// POUs/Devices/CCU/FB_METIS_CCUS
FUNCTION_BLOCK FB_METIS_CCUS
VAR_INPUT
END_VAR
VAR_OUTPUT
END_VAR
VAR
    // Cabinet Control Units (note: CCU number is not linked to the cabinet number!!!)
    ccu_ns_1 : FB_MET_CCU;
    ccu_ns_2 : FB_MET_CCU;
    // ccu_ns_3 : FB_MET_CCU; // future
    // ccu_ns_4 : FB_MET_CCU; // future
    // ccu_ns_5 : FB_MET_CCU; // future
    // ccu_ns_6 : FB_MET_CCU; // future
    
    // simulators
    // ccu_ns_1_sim : FB_SIM_MET_CCU;
    // ccu_ns_2_sim : FB_SIM_MET_CCU;
    // ccu_ns_3_sim : FB_SIM_MET_CCU;
    // ccu_ns_4_sim : FB_SIM_MET_CCU; 
    // ccu_ns_5_sim : FB_SIM_MET_CCU;
    // ccu_ns_6_sim : FB_SIM_MET_CCU;
    
    // cooling config handlers
    {attribute 'OPC.UA.DA' := '0'}
    aCoolingConfig : ARRAY[1..2] OF FB_READ_WRITE_CAB_COOLING_CONFIG;
    
    // power config handlers
    {attribute 'OPC.UA.DA' := '0'}
    aPowerConfig : ARRAY[1..2] OF FB_READ_WRITE_CAB_POWER_CONFIG;
    
    // configure bool
    {attribute 'OPC.UA.DA' := '0'}
    bConfigured : BOOL;
END_VAR

// run the cooling config handlers (before configure!)
aCoolingConfig[1](in_sName := 'Cab_Cooling_1', stConfig := ccu_ns_1.cooling.cfg);
aCoolingConfig[2](in_sName := 'Cab_Cooling_2', stConfig := ccu_ns_2.cooling.cfg);
// aCoolingConfig[3](in_sName := 'Cab_Cooling_3', stConfig := ccu_ns_3.cooling.cfg); // future
// aCoolingConfig[4](in_sName := 'Cab_Cooling_4', stConfig := ccu_ns_4.cooling.cfg); // future
// aCoolingConfig[5](in_sName := 'Cab_Cooling_5', stConfig := ccu_ns_5.cooling.cfg); // future
// aCoolingConfig[6](in_sName := 'Cab_Cooling_6', stConfig := ccu_6.cooling.cfg); // future

// run the power config handlers (before configure!)
aPowerConfig[1](in_sName := 'Cab_Power_1', stConfig := ccu_ns_1.power.cfg);
aPowerConfig[2](in_sName := 'Cab_Power_2', stConfig := ccu_ns_2.power.cfg);
// aPowerConfig[3](in_sName := 'Cab_Power_3', stConfig := ccu_ns_3.power.cfg); // future
// aPowerConfig[4](in_sName := 'Cab_Power_4', stConfig := ccu_ns_4.power.cfg); // future
// aPowerConfig[5](in_sName := 'Cab_Power_5', stConfig := ccu_ns_5.power.cfg); // future
// aPowerConfig[6](in_sName := 'Cab_Power_6', stConfig := ccu_ns_6.power.cfg); // future

// run M_Configure *after* the config handlers above! 
IF NOT bConfigured THEN
    M_Configure();
    RETURN;
END_IF


// run the CCUs
ccu_ns_1(in_sCuName := 'CCU_NS_1', in_sCabinetName := 'Cabinet 6');
ccu_ns_2(in_sCuName := 'CCU_NS_2', in_sCabinetName := 'Cabinet 4');
// ccu_ns_3(in_sCuName := 'CCU_NS_3', in_sCabinetName := 'Cabinet TBD');
// ccu_ns_4(in_sCuName := 'CCU_NS_4', in_sCabinetName := 'Cabinet TBD');
// ccu_ns_5(in_sCuName := 'CCU_NS_5', in_sCabinetName := 'Cabinet TBD');
// ccu_ns_6(in_sCuName := 'CCU_NS_6', in_sCabinetName := 'Cabinet TBD');

// run the simulators for which no hardware is available yet
// ccu_ns_3_sim(ptrDev := ADR(ccu_ns_3));
// ccu_ns_4_sim(ptrDev := ADR(ccu_ns_4)); 
// ccu_ns_5_sim(ptrDev := ADR(ccu_ns_5));
// ccu_ns_6_sim(ptrDev := ADR(ccu_ns_6));

METHOD M_Configure : BOOL
VAR_INPUT
END_VAR
VAR_INST
	{attribute 'OPC.UA.DA' := '0'}
    nConfigureState : INT;
END_VAR
VAR_IN_OUT
	//{attribute 'OPC.UA.DA' := '0'}
END_VAR
VAR
    i : INT;
    bDone : BOOL;
    iMax : INT := 2;
END_VAR

CASE nConfigureState OF
    0:  ;
        
        // start reading the configs
        FOR i := 1 TO iMax DO
            aCoolingConfig[i].M_ReadConfiguration();
            aPowerConfig[i].M_ReadConfiguration();
        END_FOR
        nConfigureState := 1;
    1:
        bDone := TRUE;
        FOR i := 1 TO iMax DO
            IF NOT aCoolingConfig[i].bReadingDoneFlag THEN
                bDone := FALSE;
			END_IF
            IF NOT aPowerConfig[i].bReadingDoneFlag THEN
                bDone := FALSE;
			END_IF
        END_FOR
        IF bDone THEN
            nConfigureState := 2;
		END_IF
    2:
        FOR i := 1 TO iMax DO
            aCoolingConfig[i].M_ClearReadingDoneFlag();
            aPowerConfig[i].M_ClearReadingDoneFlag();
        END_FOR
        bConfigured := TRUE;
        
END_CASE
END_METHOD

END_FUNCTION_BLOCK

// POUs/XML_Cfg_Read_Write/FB_READ_WRITE_CAB_COOLING_CONFIG
FUNCTION_BLOCK FB_READ_WRITE_CAB_COOLING_CONFIG EXTENDS FB_READ_WRITE_CONFIG_BASE
VAR_INPUT
	in_sName:      T_MaxString;
END_VAR
VAR_IN_OUT
	stConfig:   T_CAB_COOLING_CFG;
END_VAR

SUPER^(
    in_sEntryName  := in_sName,
    in_sSubFolder  := 'Cab_Cooling\',
    in_sXPath      := '/Cab_Cooling_Configuration/',
    in_pSymAddr    := ADR(stConfig),
    in_cbSymSize   := SIZEOF(stConfig));

END_FUNCTION_BLOCK

// POUs/XML_Cfg_Read_Write/FB_READ_WRITE_CAB_POWER_CONFIG
FUNCTION_BLOCK FB_READ_WRITE_CAB_POWER_CONFIG EXTENDS FB_READ_WRITE_CONFIG_BASE
VAR_INPUT
	in_sName:      T_MaxString;
END_VAR
VAR_IN_OUT
	stConfig:   T_CAB_POWER_CFG;
END_VAR

SUPER^(
    in_sEntryName  := in_sName,
    in_sSubFolder  := 'Cab_Power\',
    in_sXPath      := '/Cab_Power_Configuration/',
    in_pSymAddr    := ADR(stConfig),
    in_cbSymSize   := SIZEOF(stConfig));

END_FUNCTION_BLOCK

// POUs/Routines/Evacuation/FB_METIS_CRYO_EVAC
FUNCTION_BLOCK FB_METIS_CRYO_EVAC
VAR_INPUT
	in_sName:							STRING := 'EVACUATION';
	in_Cryo_Stat:					T_METIS_CRYO_STAT;
END_VAR
VAR_IN_OUT
	{attribute 'OPC.UA.DA' := '0'}
	interlocks:						T_METIS_CRYO_INTERLOCKS;
END_VAR
VAR_OUTPUT
	out_bEvacuationActive:			BOOL;
END_VAR
VAR
	// Stat
	{attribute 'TcHmiSymbol.Show'}
	stat:							T_MET_CRYO_EVACUATION_STAT;
	// Ctrl
	{attribute 'TcHmiSymbol.Show'}
	ctrl:							T_MET_CRYO_EVACUATION_CTRL;
	// Evacuation-branch A
		{attribute 'TcHmiSymbol.Show'}
	evac_branch_a:		FB_CRYO_EVAC_BRANCH_A;
	// Evacuation-branch B
		{attribute 'TcHmiSymbol.Show'}
	evac_branch_b:		FB_CRYO_EVAC_BRANCH_B;

	
	bEnable_met_evac:	BOOL;
	
	bEnable_met_evac_a:	BOOL := FALSE;
	bEnable_met_evac_b:	BOOL := FALSE;
	
	// Pressure Sensors
	sensor_VAGF1:		FB_CRYO_SENSOR_PRESSURE;	// Cryo pressure gauge VAG F1
	VAGF1:				FB_CRYO_PRESSURE_VOTE;
	sensor_VAGF2:		FB_CRYO_SENSOR_PRESSURE;	// Cryo pressure gauge VAG F2
	VAGF2:				FB_CRYO_PRESSURE_VOTE;
	sensor_VAGG1:		FB_CRYO_SENSOR_PRESSURE;	// Cryo pressure gauge VAG G1
	VAGG1:				FB_CRYO_PRESSURE_VOTE;
	sensor_VAGG2:		FB_CRYO_SENSOR_PRESSURE;	// Cryo pressure gauge VAG G2
	VAGG2:				FB_CRYO_PRESSURE_VOTE;
	VAGF:				FB_CRYO_PRESSURE_VOTE;				// Cryo pressure F
	VAGG:				FB_CRYO_PRESSURE_VOTE;				// Cryo pressure G
	
	
	// Pressure sensors IDN resistors
	
	nIdnRes_VAG_F1		AT %I* :INT;
	nIdnRes_VAG_F2		AT %I* :INT;
	nIdnRes_VAG_G1		AT %I* :INT;
	nIdnRes_VAG_G2		AT %I* :INT;
	nIdnRes_VAG_A1		AT %I* :INT;
	nIdnRes_VAG_A2		AT %I* :INT;
	nIdnRes_VAG_A3		AT %I* :INT;
	nIdnRes_VAG_B1		AT %I* :INT;
	nIdnRes_VAG_B2		AT %I* :INT;
	nIdnRes_VAG_B3		AT %I* :INT;
	
	// Pressure sensor power 24V Dig Out
	
	bPwr_VAG_F1			AT %Q* :BOOL;
	bPwr_VAG_F2         AT %Q* :BOOL;
	bPwr_VAG_G1         AT %Q* :BOOL;
	bPwr_VAG_G2         AT %Q* :BOOL;
	bPwr_VAG_A1         AT %Q* :BOOL;
	bPwr_VAG_A2         AT %Q* :BOOL;
	bPwr_VAG_A3         AT %Q* :BOOL;
	bPwr_VAG_B1         AT %Q* :BOOL;
	bPwr_VAG_B2         AT %Q* :BOOL;
	bPwr_VAG_B3         AT %Q* :BOOL;
	
	// Valve Command handling
	cmdPVVA1:			FB_CRYO_ACTUATOR_CMD;
	bCmdPVVA1:			BOOL;	// Open/Close command for PVV1
	bIntlkPVVA1:		BOOL;	// Interlock for PVV1
	
	cmdPVVB1:			FB_CRYO_ACTUATOR_CMD;
	bCmdPVVB1:			BOOL;	// Open/Close command for PVV1
	bIntlkPVVB1:		BOOL;	// Interlock for PVV1
	
//	// Valve Power
//	bBrA_PVVs_Pwr					AT %Q* :BOOL;
//	bBrA_PVVs_FeedBack_Pwr			AT %Q* :BOOL;
//	bBrB_PVVs_Pwr					AT %Q* :BOOL;
//	bBrB_PVVs_FeedBack_Pwr			AT %Q* :BOOL;
//	bPVV_Ps_Pwr						AT %Q* :BOOL;
//	bPVV_Ps_FeedBack_Pwr			AT %Q* :BOOL;
//	bPCA_PCB_VV_Pwr					AT %Q* :BOOL;
//	bPCA_PCB_VV_FeedBack_Pwr		AT %Q* :BOOL;


	// Triggers.
	//
	// Capture Enable/Disable.
	trigAutoEnable:		R_TRIG;	// bEnable_met_evac
	trigAutoDisable:	F_TRIG;	// bEnable_met_evac
	
	trigManualEnable:		R_TRIG;	// ctrl.bEnable
	trigManualDisable:		F_TRIG;	// ctrl.bEnable

	

/////////////////////////////////////////////////////////////////////////////
////////////////// Simulation////////////////////////////////////////////////
/////////////////////////////////////////////////////////////////////////////
	
	met_valves_a:		FB_SIM_MICADO_VALVES;
	met_pumps_a:		FB_SIM_MICADO_PUMPS;
	
	met_valves_b:		FB_SIM_MICADO_VALVES;
	met_pumps_b:		FB_SIM_MICADO_PUMPS;
	
	// Pressure values
	q_nVAGA1			AT %Q*:	INT := 30000;
	q_nVAGA2			AT %Q*:	INT := 30000;
	q_nVAGA3			AT %Q*:	INT := 30000;
	
	q_nVAGB1			AT %Q*:	INT := 30000;
	q_nVAGB2			AT %Q*:	INT := 30000;
	q_nVAGB3			AT %Q*:	INT := 30000;
	
	q_nVAGF1			AT %Q*:	INT := 30000;
	q_nVAGF2			AT %Q*:	INT := 30000;
	q_nVAGG1			AT %Q*:	INT := 30000;
	q_nVAGG2			AT %Q*:	INT := 30000;
	
	// 230 VAC Power  for TMPs
	
	q_bTP_A_pwr			AT %Q*: BOOL;
	bTP_A_pwr: 					BOOL := TRUE;
	q_bTP_B_pwr			AT %Q*: BOOL;
	bTP_B_pwr: 					BOOL := TRUE;
	// Dig iuput 24V source
	q_bTP_A_Ready			AT %Q*: BOOL := FALSE;
	q_bTP_A_Speed100		AT %Q*: BOOL := FALSE;
	q_bTP_A_Warning			AT %Q*: BOOL := FALSE; 
	q_bTP_A_Error			AT %Q*: BOOL := FALSE;
	q_bTP_B_Ready			AT %Q*: BOOL := FALSE;
	q_bTP_B_Speed100		AT %Q*: BOOL := FALSE;
	q_bTP_B_Warning			AT %Q*: BOOL := FALSE; 
	q_bTP_B_Error			AT %Q*: BOOL := FALSE;
	
	// Used for simulated toggle signal
	pSim:				FB_CRYO_SIM_PRESSURE;
	
	q_nCouplerState		AT %Q*:	INT := 8;

	/////////////////////
	// Cryo System logs
	/////////////////////
		
	logs:	FB_CRYO_FUNCTION_LOG;

	
	// Configure
	bConfigured:			BOOL := FALSE;
END_VAR


IF stat.bManual THEN
	;
ELSE
	IF stat.bAuto THEN
		ctrl.bEnable := bEnable_met_evac;
		stat.bAuto := FALSE;
	ELSE
		;
	END_IF
END_IF

M_Configure();

M_HandleEvents();

M_ExecuteControllers();


M_HandleInterlocks();

M_UpdateStatus();

METHOD M_AreAnyPumpsRunning : BOOL
VAR_INPUT
END_VAR


//IF  evac_branch_a.tpRef.M_GetSpeed() = 0 AND   // speed of Turbo pump on branch A
//	evac_branch_a.rpRef.M_GetSpeed() = 0 AND  // speed of roughing on branch A
//	evac_branch_b.tpRef.M_GetSpeed() = 0 AND  // speed of Turbo pump on branch B
//	evac_branch_b.rpRef.M_GetSpeed() = 0 THEN  // speed of roughing on branch B
	
//	M_AreAnyPumpsRunning := FALSE;
	
//ELSE
//	M_AreAnyPumpsRunning := TRUE;
//END_IF


M_AreAnyPumpsRunning := evac_branch_a.tpRef.M_IsRunning() OR
						evac_branch_a.rpRef.M_IsRunning() OR
						evac_branch_b.tpRef.M_IsRunning() OR
						evac_branch_b.rpRef.M_IsRunning();
END_METHOD

METHOD M_AreRoughingPumpRunning : BOOL
VAR_INPUT
END_VAR


//IF 
//	evac_branch_a.rpRef.M_GetSpeed() = 0 AND  // speed of roughing on branch A	
//	evac_branch_b.rpRef.M_GetSpeed() = 0 THEN  // speed of roughing on branch B
	
//	M_AreRoughingPumpRunning := FALSE;
	
//ELSE
//	M_AreRoughingPumpRunning := TRUE;
//END_IF

M_AreRoughingPumpRunning := evac_branch_a.rpRef.M_IsRunning() AND evac_branch_b.rpRef.M_IsRunning();
END_METHOD

METHOD M_AreTurboPumpsRunning : BOOL
VAR_INPUT
END_VAR


//IF  evac_branch_a.tpRef.M_GetSpeed() = 0 AND   // speed of Turbo pump on branch A
//	evac_branch_b.tpRef.M_GetSpeed() = 0 THEN  // speed of Turbo pump on branch B

	
//	M_AreTurboPumpsRunning := FALSE;
	
//ELSE
//	M_AreTurboPumpsRunning := TRUE;
//END_IF


M_AreTurboPumpsRunning := evac_branch_a.tpRef.M_IsRunning() AND evac_branch_a.tpRef.M_IsRunning();
END_METHOD

METHOD M_CheckBranchError : BOOL
VAR_INPUT
END_VAR
//IF  evac_branch_a.tpRef.M_GetSpeed() = 0 AND   // speed of Turbo pump on branch A
//	evac_branch_a.rpRef.M_GetSpeed() = 0 AND  // speed of roughing on branch A
//	evac_branch_b.tpRef.M_GetSpeed() = 0 AND  // speed of Turbo pump on branch B
//	evac_branch_b.rpRef.M_GetSpeed() = 0 THEN  // speed of roughing on branch B


// evac_branch_a.stat.bError
END_METHOD

METHOD M_Configure
VAR_INPUT
END_VAR
IF NOT bConfigured THEN
	

	// Enable Pressure sensor power
	bPwr_VAG_F1		 :=	TRUE;																				
	bPwr_VAG_F2      :=	TRUE;
	bPwr_VAG_G1      :=	TRUE;
	bPwr_VAG_G2      :=	TRUE;
	bPwr_VAG_A1      :=	TRUE;
	bPwr_VAG_A2      :=	TRUE;
	bPwr_VAG_A3      :=	TRUE;
	bPwr_VAG_B1      :=	TRUE;
	bPwr_VAG_B2      :=	TRUE;
	bPwr_VAG_B3      :=	TRUE;


//Enable power for valves, feedback of the valves
//	bBrA_PVVs_Pwr						:=	TRUE;	
//    bBrA_PVVs_FeedBack_Pwr	            :=	TRUE;
//    bBrB_PVVs_Pwr			            :=	TRUE;
//    bBrB_PVVs_FeedBack_Pwr	            :=	TRUE;
//    bPVV_Ps_Pwr				            :=	TRUE;
//    bPVV_Ps_FeedBack_Pwr	            :=	TRUE;
//    bPCA_PCB_VV_Pwr			            :=	TRUE;
//    bPCA_PCB_VV_FeedBack_Pwr            :=	TRUE;


	
	
	q_bTP_A_Ready	 := TRUE;
	q_bTP_A_Speed100 := TRUE;
	q_bTP_A_Warning	 := TRUE;
	q_bTP_A_Error	 := TRUE;
	q_bTP_B_Ready	 := TRUE;
	q_bTP_B_Speed100 := TRUE;
	q_bTP_B_Warning	 := TRUE;
	q_bTP_B_Error	 := TRUE;
	
// This call just configures logs at the very start.
// Logging is done by explicit calls to M_LogInfo().
logs(in_sName := in_sName);	

                                   
	bConfigured := TRUE;
END_IF
END_METHOD

METHOD M_ExecuteControllers
VAR_INPUT
END_VAR

// 230 VAC Power  for TMPs

	q_bTP_A_pwr := bTP_A_pwr;
    q_bTP_B_pwr := bTP_B_pwr;

// METIS Cryostat pressures
sensor_VAGF1(in_sName := 'VAGF1' ,in_nType := E_CRYO_SENSOR_TYPE_PRESS.PKR_360,	in_nSampleTime := 100);
sensor_VAGF2(in_sName := 'VAGF2' ,in_nType := E_CRYO_SENSOR_TYPE_PRESS.PKR_360,	in_nSampleTime := 100);
sensor_VAGG1(in_sName := 'VAGG1' ,in_nType := E_CRYO_SENSOR_TYPE_PRESS.PKR_360,	in_nSampleTime := 100);
sensor_VAGG2(in_sName := 'VAGG2' ,in_nType := E_CRYO_SENSOR_TYPE_PRESS.PKR_360,	in_nSampleTime := 100);


ctrl.por_VAGF1(in_bEnable := ctrl.bSim_Press_VAGF1);	// Simulation flag override
VAGF1(
	in_sName		:= 'VAGF1',
	in_bSimulation	:= ctrl.por_VAGF1.out_bEnable,
	in_nNumSensor	:= 1,
	in_nVoteMethod	:= E_CRYO_VOTE.V_AVE,
	in_pSensor1		:= ADR(sensor_VAGF1));

ctrl.por_VAGF2(in_bEnable := ctrl.bSim_Press_VAGF2);	// Simulation flag override
VAGF2(
	in_sName		:= 'VAGF2',
	in_bSimulation	:= ctrl.por_VAGF2.out_bEnable,
	in_nNumSensor	:= 1,
	in_nVoteMethod	:= E_CRYO_VOTE.V_AVE,
	in_pSensor1		:= ADR(sensor_VAGF2));

ctrl.por_VAGG1(in_bEnable := ctrl.bSim_Press_VAGG1);	// Simulation flag override
VAGG1(
	in_sName		:= 'VAGG1',
	in_bSimulation	:= ctrl.por_VAGG1.out_bEnable,
	in_nNumSensor	:= 1,
	in_nVoteMethod	:= E_CRYO_VOTE.V_AVE,
	in_pSensor1		:= ADR(sensor_VAGG1));

ctrl.por_VAGG2(in_bEnable := ctrl.bSim_Press_VAGG2);	// Simulation flag override
VAGG2(
	in_sName		:= 'VAGG2',
	in_bSimulation	:= ctrl.por_VAGG2.out_bEnable,
	in_nNumSensor	:= 1,
	in_nVoteMethod	:= E_CRYO_VOTE.V_AVE,
	in_pSensor1		:= ADR(sensor_VAGG2));

ctrl.por_VAGF(in_bEnable := ctrl.bSim_Press_VAGF);	// Simulation flag override
VAGF(
	in_sName		:= 'VAGF',
	in_bSimulation	:= ctrl.por_VAGF.out_bEnable,
	in_nNumSensor	:= 2,
	in_nVoteMethod	:= E_CRYO_VOTE.V_1oo2,
	in_pSensor1		:= ADR(sensor_VAGF1),
	in_pSensor2		:= ADR(sensor_VAGF2));
	
ctrl.por_VAGG(in_bEnable := ctrl.bSim_Press_VAGG);	// Simulation flag override
VAGG(
	in_sName		:= 'VAGG',
	in_bSimulation	:= ctrl.por_VAGG.out_bEnable,
	in_nNumSensor	:= 2,
	in_nVoteMethod	:= E_CRYO_VOTE.V_1oo2,
	in_pSensor1		:= ADR(sensor_VAGG1),
	in_pSensor2		:= ADR(sensor_VAGG2));
	
	
	
	
	
	
	
	
	

	
// METIS evacuation system
cmdPVVA1(in_bEnable:=bCmdPVVA1,in_bInterlock:=bIntlkPVVA1);	// Handling of PVV1 commands
cmdPVVB1(in_bEnable:=bCmdPVVB1,in_bInterlock:=bIntlkPVVB1);	// Handling of PVV1 commands


IF ctrl.bEnable THEN
	bEnable_met_evac_a := TRUE;
	bEnable_met_evac_b := TRUE;
ELSE
	bEnable_met_evac_a := FALSE;
	bEnable_met_evac_b := FALSE;
END_IF

evac_branch_a(
	in_bEnable		:= bEnable_met_evac_a,
	in_RefVAGF		:= VAGF, 
	in_RefVAGG		:= VAGG);

evac_branch_b(
	in_bEnable		:= bEnable_met_evac_a,
	in_RefVAGF		:= VAGF, 
	in_RefVAGG		:= VAGG);
	
	
	
{IF defined (V2_SIM)}
	{info 'Simulated valves'}	

pSim();	// Just to have a simulated Toggle signal.

// Simulation of METIS valves
met_valves_a();
met_valves_b();	

// Simulation of METIS pumps
met_pumps_a(in_RefPVP:=evac_branch_a.rp, in_RefTMP:=evac_branch_a.tp);	
met_pumps_b(in_RefPVP:=evac_branch_b.rp, in_RefTMP:=evac_branch_b.tp);	

{END_IF}
END_METHOD

METHOD M_HandleEvents
VAR_INPUT
END_VAR
VAR_INST
    nEvacOnOffState : UINT := 0; // 0=Idle, 10=AutoOn, 20=AutoOff, 30=ManualOn, 40=ManualOff
END_VAR

trigAutoEnable    (CLK := bEnable_met_evac);
trigAutoDisable   (CLK := bEnable_met_evac); 

trigManualEnable  (CLK := ctrl.bEnable);
trigManualDisable (CLK := ctrl.bEnable);


CASE nEvacOnOffState OF

    0: // Idle / waiting for an event
        IF trigAutoEnable.Q THEN
            nEvacOnOffState := 10;
        ELSIF trigAutoDisable.Q THEN
            nEvacOnOffState := 20;
        ELSIF trigManualEnable.Q THEN
            nEvacOnOffState := 30;
        ELSIF trigManualDisable.Q THEN
            nEvacOnOffState := 40;
        END_IF

    10: // Auto Enable event
        stat.sState := 'EVACUATION started automatically';
        logs.M_LogInfo('EVACUATION started automatically');
		M_ResetValves();
        nEvacOnOffState := 0; // back to idle

    20: // Auto Disable event
        stat.sState := 'EVACUATION stopped automatically';
        logs.M_LogInfo('EVACUATION stopped automatically');
		M_ResetValves();
        nEvacOnOffState := 0;

    30: // Manual Enable event
        stat.sState := 'EVACUATION started by operator';
        logs.M_LogInfo('EVACUATION started by operator');
		M_ResetValves();
        nEvacOnOffState := 0;

    40: // Manual Disable event
        stat.sState := 'EVACUATION interrupted by operator';
        logs.M_LogInfo('EVACUATION interrupted by operator');
		M_ResetValves();
        nEvacOnOffState := 0;

END_CASE
END_METHOD

METHOD M_HandleInterlocks
VAR_INPUT
END_VAR
END_METHOD

METHOD M_ResetValves : BOOL
VAR_INPUT
END_VAR
evac_branch_a.M_ResetValves();
evac_branch_b.M_ResetValves();
END_METHOD

METHOD M_SetAuto : BOOL
VAR_INPUT
END_VAR
stat.bAuto := TRUE;
END_METHOD

METHOD PRIVATE M_SetError
VAR_INPUT
    nCode     : UDINT;
    sMessage  : STRING;
END_VAR


stat.Error.nCode := nCode;
stat.Error.sMessage := sMessage;
stat.bError := TRUE;
//stat.nState := E_MET_CRYO_EVA.ERROR;
END_METHOD

METHOD M_Start_Evacuation : BOOL
VAR_INPUT
END_VAR
stat.bAuto := TRUE;
bEnable_met_evac := TRUE;
END_METHOD

METHOD M_Stop_Evacuation : BOOL
VAR_INPUT
END_VAR

stat.bAuto := TRUE;
bEnable_met_evac := FALSE;
END_METHOD

METHOD M_UpdateStatus
VAR_INPUT
END_VAR


// Check Pre-Conditions for HMI Enable 

stat.bPreConditionsMet :=  in_Cryo_Stat.bVentingValvesAreClosed;


stat.bActive := ctrl.bEnable;
out_bEvacuationActive := stat.bActive;

stat.bBusy := stat.bActive;
stat.bDone := NOT stat.bActive;
END_METHOD

END_FUNCTION_BLOCK

// POUs/Routines/Evacuation/FB_CRYO_EVAC_BRANCH_A
FUNCTION_BLOCK FB_CRYO_EVAC_BRANCH_A EXTENDS FB_CRYO_EVAC_BASE_50000
VAR_INPUT
END_VAR
VAR_OUTPUT
END_VAR
VAR
	// Specify pumps
	{attribute 'TcHmiSymbol.Show'}
	rp:				FB_CRYO_PUMP_ECODRY;	// Roughing Pump
	{attribute 'TcHmiSymbol.Show'}
	tp:				FB_CRYO_PUMP_ATH2303M;	// Turbomolecular Pump
	
	// Pumps command handeling
	cor_rp:			FB_CRYO_CMD_OVERRIDE;
	cor_tp:			FB_CRYO_CMD_OVERRIDE;
	
	
	
	bReset_Valves:		BOOL:= FALSE;
	
	
END_VAR






SUPER^();	// Execute base FB code.

IF bReset_Valves THEN
	M_ResetValves();
	bReset_Valves := FALSE;
END_IF

METHOD M_Configure
VAR_INPUT
END_VAR
//
// Specific METIS configuration.
//
IF NOT stat.bConfigured	THEN
	//
	// MANDATORY !!!
	// Call base FB::M_Configure() to set the pointers.
	//
	SUPER^.M_Configure();
	

	// MANDATORY: Set References for pumps!!!
	// If not done, system will crash !!!
	rpRef	REF=rp;
	tpRef	REF=tp;
	

	// Specific instance configuration, e.g. anything different
	// from the default values given in the cfg structure of type T_CRYO_EVAC_CFG_50000.
	cfg.nType_VAG1	:= E_CRYO_SENSOR_TYPE_PRESS.PKR_360;
	cfg.nType_VAG2	:= E_CRYO_SENSOR_TYPE_PRESS.PKR_360;
	cfg.nType_VAG3	:= E_CRYO_SENSOR_TYPE_PRESS.PKR_360;
	
	cfg.nType_VAGF1	:= E_CRYO_SENSOR_TYPE_PRESS.PKR_360;
	cfg.nType_VAGF2	:= E_CRYO_SENSOR_TYPE_PRESS.PKR_360;
	cfg.nType_VAGG1	:= E_CRYO_SENSOR_TYPE_PRESS.PKR_360;
	cfg.nType_VAGG2	:= E_CRYO_SENSOR_TYPE_PRESS.PKR_360;
	
	// Prevacuum pressure threshold [mbar]: TMP start below this 
	
	cfg.lrThld_Prevac:= 0.5;	 	

// Reseting all valves. Without this, the valves were not initializing in error and were unable to recover
	PVV1.M_Reset();
	PVV2.M_Reset();
	PVV3.M_Reset();
	PVV4.M_Reset();
	GBV.M_Reset();
	
	
	stat.bConfigured	:= TRUE;
ELSE
	RETURN;	// Nothing to do any more
END_IF
END_METHOD

METHOD M_ExecuteControllers
VAR_INPUT
END_VAR
// Pumps command overide 

cor_rp(in_bEnable:= ctrl.bEnable_PVP);
cor_tp(in_bEnable:= ctrl.bEnable_TMP);


{IF defined (V2_SIM)}
	{info 'Simulated Pumps'}
	
		// Roughing Pump	
	rp(	
		in_bSimulation	:= TRUE,
		in_sName		:= 'ECODRY A',
		in_bEnable		:= cor_rp.out_bEnable,
		in_nSlaveID		:= 1,
		in_sVersion		:= 'V22',
		in_nPeriod		:= 2000,
		in_bFeedbackActiveLow := TRUE			// TRUE for simulation and FALSE for real hardware		
	);
	
	// Turbo Molecular Pump
	tp(	
		in_bSimulation	:= TRUE,
		in_sName		:= 'ATH2303M A',
		in_bEnable		:= cor_tp.out_bEnable,
		in_nModel		:= 2303,
		in_bAutoMonitor	:= TRUE,
		in_nPeriod		:= 2000);
{END_IF}



{IF defined (V1_HW)}
	{info 'Actual Pumps are Active'}
	
		// Roughing Pump	
	rp(	
		in_bSimulation	:= FALSE,
		in_sName		:= 'ECODRY A',
		in_bEnable		:= cor_rp.out_bEnable,
		in_nSlaveID		:= 1,
		in_sVersion		:= 'V22',
		in_nPeriod		:= 2000,
		in_bFeedbackActiveLow := FALSE			// TRUE for simulation and FALSE for real hardware		
	);
	
	// Turbo Molecular Pump
	tp(	
		in_bSimulation	:= FALSE,
		in_sName		:= 'ATH2303M A',
		in_bEnable		:= cor_tp.out_bEnable,
		in_nModel		:= 2303,
		in_bAutoMonitor	:= TRUE,
		in_nPeriod		:= 2000);

{END_IF}





SUPER^.M_ExecuteControllers();
END_METHOD

METHOD M_HandleInterlocks
VAR_INPUT
END_VAR
////////////////////////////////////////////////////////////////////
// IMPORTANT NOTE !!!
//
// The naming of valves and pumps is in accordance with
// the official ESO document 
// Sequences for vacuum vessel 2500 - 50000L by Marcus v5.pdf.
//
// MICADO names are different/swapped.
//
/////////////////////////////////////////////////////////////////////


///////////////////////////////////////////
// Translation Table MICADO --> ESO Naming
///////////////////////////////////////////
(*
MPA-A-PVP	PVP
MPA-A-TMP	TMP

MPA-A-GBV	GBV
MPA-A-PVV1	PVV3
MPA-A-PVV2	PVV4
MPA-A-PVV3	PVV1
MPA-A-PVV4	PVV2

TMPA-A-VAG1	VAG3
TMPA-A-VAG2	VAG2
TMPA-A-VAG3	VAG1

WRGA-A-VAG	VAGF
WRGA-B-VAG	VAGG
*)


//////////////////////////////////////////
////////////     VALVES       ////////////
//////////////////////////////////////////


//				
// TMPA-A-GBV: Can only be opened IF TMPA-A-PVP is ON.
//----------------------------------------
// GBV: Can only be opened IF PVP is ON.
//
IF rp.stat.bMoving	THEN
	ctrl.cor_GBV.M_SetAllPermitted();			// OPEN/CLOSE allowed.
ELSE
	ctrl.cor_GBV.M_SetPermissions(FALSE,TRUE);	// Only CLOSE allowed.
END_IF


//
// TMPA-A-PVV3: Can only be opened if:
// 	i. TMPA-A-VAG1 is less than 10-1 mbar
// 	ii. TMPA-A-TMP is OFF
// 	iii. WRGA-A-VAG and WRGA-B-VAG show pressure readings greater than 10-1 mbar.
//----------------------------------------
// PVV1: Can only be opened if:
// 	i. VAG3 is less than 10-1 mbar
// 	ii. TMP is OFF
// 	iii. VAGF and VAGG show pressure readings greater than 10-1 mbar.
//
IF	VAG3.stat.lrPressure < 0.1  AND  
	NOT tp.stat.bSpeed100  		AND 
	VAGF.stat.lrPressure > 0.1  AND 
	VAGG.stat.lrPressure > 0.1		THEN
	ctrl.cor_PVV1.M_SetAllPermitted();			// OPEN/CLOSE allowed.
ELSE
	ctrl.cor_PVV1.M_SetPermissions(FALSE,TRUE);	// Only CLOSE allowed.
END_IF


//
//	TMPA-A-PVV4: Can only be opened if:
// 	i. TMPA-A-VAG1 and TMPA-A-VAG3 show pressure readings of less than 10-1mbar
// 	ii. TMPA-A-TMP is OFF
// 	iii. WRGA-A-VAG and WRGA-B-VAG show pressure readings greater than 10-1mbar.
//----------------------------------------
//	PVV2: Can only be opened if:
// 	i. TMPA-A-VAG3 and TMPA-A-VAG1 show pressure readings of less than 10-1 mbar
// 	ii. TMP is OFF
// 	iii. VAGF and VAGG show pressure readings greater than 10-1 mbar.
//
IF	VAG3.stat.lrPressure < 0.1  AND  
	VAG1.stat.lrPressure < 0.1  AND  
	NOT tp.stat.bSpeed100  		AND 
	VAGF.stat.lrPressure > 0.1  AND 
	VAGG.stat.lrPressure > 0.1		THEN
	ctrl.cor_PVV2.M_SetAllPermitted();			// OPEN/CLOSE allowed.
ELSE
	ctrl.cor_PVV2.M_SetPermissions(FALSE,TRUE);	// Only CLOSE allowed.
END_IF


//
// TMPA-A-PVV1: Can only be opened if TMPA-A-TMP is ON or TMPA-A-PVV2 is closed.
//----------------------------------------
// PVV3: Can only be opened if TMP is ON or PVV4 is closed.
//
IF tp.stat.bSpeed100  OR  PVV4.stat.bActOFF	THEN
	ctrl.cor_PVV3.M_SetAllPermitted();			// OPEN/CLOSE allowed.
ELSE
	ctrl.cor_PVV3.M_SetPermissions(FALSE,TRUE);	// Only CLOSE allowed.
END_IF


//
// TMPA-A-PVV2: Can only be opened if TMPA-A-VAG1 and TMPA-A-VAG2 show pressure readings below 10-1 mbar
//----------------------------------------
// PVV4: Can only be opened if VAG3 and VAG2 show pressure readings below 10-1 mbar
//
IF VAG3.stat.lrPressure < 0.1  AND  VAG2.stat.lrPressure < 0.1	THEN
	ctrl.cor_PVV4.M_SetAllPermitted();			// OPEN/CLOSE allowed.
ELSE
	ctrl.cor_PVV4.M_SetPermissions(FALSE,TRUE);	// Only CLOSE allowed.
END_IF



//////////////////////////////////////////
////////////     PUMPS        ////////////
//////////////////////////////////////////


//
// TMPA-A-PVP: No interlock.
//----------------------------------------
// PVP: No interlock.
//
ctrl.cor_PVP.M_SetAllPermitted();	// ON/OFF allowed.


//
// TMPA-A-TMP: Can only be switched ON if WRGA-A-VAG and WRGA-B-VAG show pressure readings below 10-1 mbar
//----------------------------------------
// TMP: Can only be switched ON if VAGF and VAGG show pressure readings below 10-1 mbar
//
IF	VAGF.stat.lrPressure < (0.1 + cfg.lrThld_PrevacTol) AND 
	VAGG.stat.lrPressure < (0.1 + cfg.lrThld_PrevacTol)		THEN
	ctrl.cor_TMP.M_SetAllPermitted();			// ON/OFF allowed.
ELSE
	ctrl.cor_TMP.M_SetPermissions(FALSE,TRUE);	// Only OFF allowed.
END_IF
END_METHOD

METHOD M_ResetValves
VAR_INPUT
END_VAR
PVV1.M_Reset();
PVV2.M_Reset();
PVV3.M_Reset();
PVV4.M_Reset();
GBV.M_Reset();
END_METHOD

END_FUNCTION_BLOCK

// POUs/Routines/Evacuation/FB_CRYO_EVAC_BRANCH_B
FUNCTION_BLOCK FB_CRYO_EVAC_BRANCH_B EXTENDS FB_CRYO_EVAC_BASE_50000
VAR_INPUT
END_VAR
VAR_OUTPUT
END_VAR
VAR
	// Specify pumps
	{attribute 'TcHmiSymbol.Show'}
	rp:				FB_CRYO_PUMP_ECODRY;	// Roughing Pump
	{attribute 'TcHmiSymbol.Show'}
	tp:				FB_CRYO_PUMP_ATH2303M;	// Turbomolecular Pump
	
	// Pumps command handeling
	cor_rp:			FB_CRYO_CMD_OVERRIDE;
	cor_tp:			FB_CRYO_CMD_OVERRIDE;
	
	
		bReset_Valves:		BOOL:= FALSE;
		
END_VAR

SUPER^();	// Execute base FB code.

IF bReset_Valves THEN
	M_ResetValves();
	bReset_Valves := FALSE;
END_IF

METHOD M_Configure
VAR_INPUT
END_VAR
//
// Specific MICADO configuration.
//
IF NOT stat.bConfigured	THEN
	//
	// MANDATORY !!!
	// Call base FB::M_Configure() to set the pointers.
	//
	SUPER^.M_Configure();
	

	// MANDATORY: Set References for pumps!!!
	// If not done, system will crash !!!
	rpRef	REF=rp;
	tpRef	REF=tp;
	

	// Specific instance configuration, e.g. anything different
	// from the default values given in the cfg structure of type T_CRYO_EVAC_CFG_50000.
	cfg.nType_VAG1	:= E_CRYO_SENSOR_TYPE_PRESS.PKR_360;
	cfg.nType_VAG2	:= E_CRYO_SENSOR_TYPE_PRESS.PKR_360;
	cfg.nType_VAG3	:= E_CRYO_SENSOR_TYPE_PRESS.PKR_360;
	cfg.nType_VAGF1	:= E_CRYO_SENSOR_TYPE_PRESS.PKR_360;
	cfg.nType_VAGF2	:= E_CRYO_SENSOR_TYPE_PRESS.PKR_360;
	cfg.nType_VAGG1	:= E_CRYO_SENSOR_TYPE_PRESS.PKR_360;
	cfg.nType_VAGG2	:= E_CRYO_SENSOR_TYPE_PRESS.PKR_360;
	
	// Prevacuum pressure threshold [mbar]: TMP start below this 
	
	cfg.lrThld_Prevac:= 0.5;	 

// Reseting all valves. Without this, the valves were not initializing in error and were unable to recover
	PVV1.M_Reset();
	PVV2.M_Reset();
	PVV3.M_Reset();
	PVV4.M_Reset();
	GBV.M_Reset();
	
	stat.bConfigured	:= TRUE;
ELSE
	RETURN;	// Nothing to do any more
END_IF
END_METHOD

METHOD M_ExecuteControllers
VAR_INPUT
END_VAR
// Pumps command overide 

cor_rp(in_bEnable:= ctrl.bEnable_PVP);
cor_tp(in_bEnable:= ctrl.bEnable_TMP);


{IF defined (V2_SIM)}
	{info 'Simulated Pumps'}
	
		// Roughing Pump	
	rp(	
		in_bSimulation	:= TRUE,
		in_sName		:= 'ECODRY B',
		in_bEnable		:= cor_rp.out_bEnable,
		in_nSlaveID		:= 1,
		in_sVersion		:= 'V22',
		in_nPeriod		:= 2000,
		in_bFeedbackActiveLow := TRUE			// TRUE for simulation and FALSE for real hardware		
	);
	
	// Turbo Molecular Pump
	tp(	
		in_bSimulation	:= TRUE,
		in_sName		:= 'ATH2303M B',
		in_bEnable		:= cor_tp.out_bEnable,
		in_nModel		:= 2303,
		in_bAutoMonitor	:= TRUE,
		in_nPeriod		:= 2000);
{END_IF}



{IF defined (V1_HW)}
	{info 'Actual Pumps are Active'}
	
		// Roughing Pump	
	rp(	
		in_bSimulation	:= FALSE,
		in_sName		:= 'ECODRY B',
		in_bEnable		:= cor_rp.out_bEnable,
		in_nSlaveID		:= 1,
		in_sVersion		:= 'V22',
		in_nPeriod		:= 2000,
		in_bFeedbackActiveLow := FALSE			// TRUE for simulation and FALSE for real hardware		
	);
	
	// Turbo Molecular Pump
	tp(	
		in_bSimulation	:= FALSE,
		in_sName		:= 'ATH2303M B',
		in_bEnable		:= cor_tp.out_bEnable,
		in_nModel		:= 2303,
		in_bAutoMonitor	:= TRUE,
		in_nPeriod		:= 2000);

{END_IF}





SUPER^.M_ExecuteControllers();
END_METHOD

METHOD M_HandleInterlocks
VAR_INPUT
END_VAR
////////////////////////////////////////////////////////////////////
// IMPORTANT NOTE !!!
//
// The naming of valves and pumps is in accordance with
// the official ESO document 
// Sequences for vacuum vessel 2500 - 50000L by Marcus v5.pdf.
//
// MICADO names are different/swapped.
//
/////////////////////////////////////////////////////////////////////


///////////////////////////////////////////
// Translation Table MICADO --> ESO Naming
///////////////////////////////////////////
(*
MPA-A-PVP	PVP
MPA-A-TMP	TMP

MPA-A-GBV	GBV
MPA-A-PVV1	PVV3
MPA-A-PVV2	PVV4
MPA-A-PVV3	PVV1
MPA-A-PVV4	PVV2

TMPA-A-VAG1	VAG3
TMPA-A-VAG2	VAG2
TMPA-A-VAG3	VAG1

WRGA-A-VAG	VAGF
WRGA-B-VAG	VAGG
*)


//////////////////////////////////////////
////////////     VALVES       ////////////
//////////////////////////////////////////


//				
// TMPA-A-GBV: Can only be opened IF TMPA-A-PVP is ON.
//----------------------------------------
// GBV: Can only be opened IF PVP is ON.
//
IF rp.stat.bMoving	THEN
	ctrl.cor_GBV.M_SetAllPermitted();			// OPEN/CLOSE allowed.
ELSE
	ctrl.cor_GBV.M_SetPermissions(FALSE,TRUE);	// Only CLOSE allowed.
END_IF


//
// TMPA-A-PVV3: Can only be opened if:
// 	i. TMPA-A-VAG1 is less than 10-1 mbar
// 	ii. TMPA-A-TMP is OFF
// 	iii. WRGA-A-VAG and WRGA-B-VAG show pressure readings greater than 10-1 mbar.
//----------------------------------------
// PVV1: Can only be opened if:
// 	i. VAG3 is less than 10-1 mbar
// 	ii. TMP is OFF
// 	iii. VAGF and VAGG show pressure readings greater than 10-1 mbar.
//
IF	VAG3.stat.lrPressure < 0.1  AND  
	NOT tp.stat.bSpeed100  		AND 
	VAGF.stat.lrPressure > 0.1  AND 
	VAGG.stat.lrPressure > 0.1		THEN
	ctrl.cor_PVV1.M_SetAllPermitted();			// OPEN/CLOSE allowed.
ELSE
	ctrl.cor_PVV1.M_SetPermissions(FALSE,TRUE);	// Only CLOSE allowed.
END_IF


//
//	TMPA-A-PVV4: Can only be opened if:
// 	i. TMPA-A-VAG1 and TMPA-A-VAG3 show pressure readings of less than 10-1mbar
// 	ii. TMPA-A-TMP is OFF
// 	iii. WRGA-A-VAG and WRGA-B-VAG show pressure readings greater than 10-1mbar.
//----------------------------------------
//	PVV2: Can only be opened if:
// 	i. TMPA-A-VAG3 and TMPA-A-VAG1 show pressure readings of less than 10-1 mbar
// 	ii. TMP is OFF
// 	iii. VAGF and VAGG show pressure readings greater than 10-1 mbar.
//
IF	VAG3.stat.lrPressure < 0.1  AND  
	VAG1.stat.lrPressure < 0.1  AND  
	NOT tp.stat.bSpeed100  		AND 
	VAGF.stat.lrPressure > 0.1  AND 
	VAGG.stat.lrPressure > 0.1		THEN
	ctrl.cor_PVV2.M_SetAllPermitted();			// OPEN/CLOSE allowed.
ELSE
	ctrl.cor_PVV2.M_SetPermissions(FALSE,TRUE);	// Only CLOSE allowed.
END_IF


//
// TMPA-A-PVV1: Can only be opened if TMPA-A-TMP is ON or TMPA-A-PVV2 is closed.
//----------------------------------------
// PVV3: Can only be opened if TMP is ON or PVV4 is closed.
//
IF tp.stat.bSpeed100  OR  PVV4.stat.bActOFF	THEN
	ctrl.cor_PVV3.M_SetAllPermitted();			// OPEN/CLOSE allowed.
ELSE
	ctrl.cor_PVV3.M_SetPermissions(FALSE,TRUE);	// Only CLOSE allowed.
END_IF


//
// TMPA-A-PVV2: Can only be opened if TMPA-A-VAG1 and TMPA-A-VAG2 show pressure readings below 10-1 mbar
//----------------------------------------
// PVV4: Can only be opened if VAG3 and VAG2 show pressure readings below 10-1 mbar
//
IF VAG3.stat.lrPressure < 0.1  AND  VAG2.stat.lrPressure < 0.1	THEN
	ctrl.cor_PVV4.M_SetAllPermitted();			// OPEN/CLOSE allowed.
ELSE
	ctrl.cor_PVV4.M_SetPermissions(FALSE,TRUE);	// Only CLOSE allowed.
END_IF



//////////////////////////////////////////
////////////     PUMPS        ////////////
//////////////////////////////////////////


//
// TMPA-A-PVP: No interlock.
//----------------------------------------
// PVP: No interlock.
//
ctrl.cor_PVP.M_SetAllPermitted();	// ON/OFF allowed.


//
// TMPA-A-TMP: Can only be switched ON if WRGA-A-VAG and WRGA-B-VAG show pressure readings below 10-1 mbar
//----------------------------------------
// TMP: Can only be switched ON if VAGF and VAGG show pressure readings below 10-1 mbar
//
IF	VAGF.stat.lrPressure < (0.1 + cfg.lrThld_PrevacTol) AND 
	VAGG.stat.lrPressure < (0.1 + cfg.lrThld_PrevacTol)		THEN
	ctrl.cor_TMP.M_SetAllPermitted();			// ON/OFF allowed.
ELSE
	ctrl.cor_TMP.M_SetPermissions(FALSE,TRUE);	// Only OFF allowed.
END_IF
END_METHOD

METHOD M_ResetValves
VAR_INPUT
END_VAR
PVV1.M_Reset();
PVV2.M_Reset();
PVV3.M_Reset();
PVV4.M_Reset();
GBV.M_Reset();
END_METHOD

END_FUNCTION_BLOCK

// POUs/Routines/Venting/FB_METIS_CRYO_VENTING
FUNCTION_BLOCK FB_METIS_CRYO_VENTING
VAR_INPUT
	in_sName:						STRING := 'VENTING';
	in_Cryo_Stat:					T_METIS_CRYO_STAT;
	//in_bEnable:		BOOL := FALSE;	// System active while in_bEnable is TRUE
	in_RefVAGF:		REFERENCE TO FB_CRYO_PRESSURE_VOTE;
	in_RefVAGG:		REFERENCE TO FB_CRYO_PRESSURE_VOTE;

END_VAR
VAR_IN_OUT
	{attribute 'OPC.UA.DA' := '0'}
	interlocks:						T_METIS_CRYO_INTERLOCKS;
END_VAR
VAR_OUTPUT
	out_bVentingActive:		BOOL := FALSE;
END_VAR
VAR
	// Venting Valves
	N2V_1:		FB_CRYO_VALVE_CTRL;		// Venting valve 1
	N2V_2:		FB_CRYO_VALVE_CTRL;		// venting valve 2
	
	
	// Pointers to valves
	ptrV:	ARRAY [1..2] OF POINTER TO FB_CRYO_VALVE_CTRL;
	// Pointers to valve commands
	ptrVC:	ARRAY [1..2] OF POINTER TO FB_CRYO_CMD_OVERRIDE;
	// Pointers to Enable flags for valves
	ptrEV:	ARRAY [1..2] OF POINTER TO BOOL;	
	
	cmdN2V_1:	FB_CRYO_ACTUATOR_CMD;	// Handling of Valve1 command
	cmdN2V_2:	FB_CRYO_ACTUATOR_CMD;	// Handling of Valve1 command
	
	// System commands for Valve1 and Valve2
	
	
	////////////
	// Pressure
	////////////
	
	// Pressure transducers
	{attribute 'OPC.UA.DA' := '1'}	
	sensor_HPG1:	FB_CRYO_SENSOR_PRESSURE;	// High pressure gauge #1
	{attribute 'OPC.UA.DA' := '1'}
	sensor_HPG2:	FB_CRYO_SENSOR_PRESSURE;	// High pressure gauge #2
	
	// Pressure sensors IDN resistors
	nIdnRes_HPG1		AT %I* :INT;
	nIdnRes_HPG2		AT %I* :INT;
	
	// Pressure sensor power 24V Dig Out
	bPwr_HPG1			AT %Q* :BOOL;
	bPwr_HPG2			AT %Q* :BOOL;
	
	// Pressure measurements
	{attribute 'OPC.UA.DA' := '1'}
	HPG1:	FB_CRYO_PRESSURE_VOTE;				// High pressure
	{attribute 'OPC.UA.DA' := '1'}
	HPG2:	FB_CRYO_PRESSURE_VOTE;				// High pressure
	{attribute 'OPC.UA.DA' := '1'}
	HPG:	FB_CRYO_PRESSURE_VOTE;				// High pressure
	
	//	
	
	cfg:	T_MET_CRYO_VENTING_CFG;
	ctrl:	T_MET_CRYO_VENTING_CTRL;
	stat:	T_MET_CRYO_VENTING_STAT;
	
	
	timer:	TON;
	trig:	R_TRIG;	// Start trigger
	
	// GUI staff
	guiValveIndex:	UINT := 1;	// Index for Valve Engineering GUI
	
	// Configure
	bConfigured:		BOOL := FALSE;	
	bReset_Valves:		BOOL:= FALSE;
	
	
		//
	// Triggers.
	//
	// Capture Enable/Disable.
	trigEnable:		R_TRIG;	// in_bEnable
	trigDisable:	F_TRIG;	// in_bEnable
	
	// Capture Venting pressure ahieved
	trigVentingPressureAchieved:	R_TRIG;
	
	// Simulation HPG pressure sensors
	
	// Pressure values
	q_nSimHPG1			AT %Q*:	INT := 30000;
	q_nSimHPG2			AT %Q*:	INT := 30000;
	
	/////////////////////
	// Cryo System logs
	/////////////////////
		
	logs:	FB_CRYO_FUNCTION_LOG;
	
	
END_VAR
VAR CONSTANT

    // --- [4000] Preconditions ---
    E4000_VacuumPumpsStillRunning                 : UDINT := 4000001; // One or more vacuum pumps are still running
    E4001_TemperatureBelow280K                    : UDINT := 4000002; // One or more cryostat temperatures are below 280 K
    E4002_LN2RefillingActive                      : UDINT := 4000003; // LN2 refilling is still active
    E4003_RegenerationActive                      : UDINT := 4000004; // Sorption pump regeneration is still active
    E4004_GN2HoseNotConnected                     : UDINT := 4000005; // GN2 hose is not connected
    E4005_VentingAlreadyActive                    : UDINT := 4000006; // Venting requested while already active

    // --- [4100] Valve and Actuator Errors ---
    E4100_VentingValve1_FailedToOpen              : UDINT := 4100001; // Venting valve 1 failed to open
    E4101_VentingValve2_FailedToOpen              : UDINT := 4100002; // Venting valve 2 failed to open
    E4102_VentingValve1_FailedToClose             : UDINT := 4100003; // Venting valve 1 failed to close
    E4103_VentingValve2_FailedToClose             : UDINT := 4100004; // Venting valve 2 failed to close
    E4104_VentingValveStateConflict               : UDINT := 4100005; // Venting valves not in expected configuration
    E4105_CoolersStillRunning                     : UDINT := 4100006; // One or more coolers are still running at venting start

    // --- [4200] Pressure Monitoring Errors ---
    E4200_HPG_PressureTooHigh                     : UDINT := 4200001; // HPG pressure > ambient pressure + 50 mbar
    E4201_HPG_PressureSensorFault                 : UDINT := 4200002; // HPG pressure sensor invalid or faulty
    E4202_HPG_PressureNotRising                   : UDINT := 4200003; // HPG pressure not increasing after venting started
    E4203_HPG_PressureRiseTooFast                 : UDINT := 4200004; // HPG pressure increasing too fast during venting
    E4204_HPG_PressureDidNotReachTarget           : UDINT := 4200005; // HPG pressure did not reach ambient + 50 mbar within allowed time

    // --- [4300] Sequence Timing Errors ---
    E4300_VentingStartTimeout                     : UDINT := 4300001; // Venting sequence did not start within allowed time
    E4301_VentingDurationTimeout                  : UDINT := 4300002; // Venting exceeded maximum allowed duration
    E4302_VentingValveOpenTimeout                 : UDINT := 4300003; // Timeout while opening venting valves
    E4303_VentingValveCloseTimeout                : UDINT := 4300004; // Timeout while closing venting valves

    // --- [4400] Manual Intervention / Abort ---
    E4400_OperatorAbortedVenting                  : UDINT := 4400001; // Operator manually stopped venting
    E4401_OperatorClosedVentingValves             : UDINT := 4400002; // Operator manually closed venting valves during venting

    // --- [4500] Interlock Violations ---
    E4500_VacuumPumpsStartedDuringVenting         : UDINT := 4500001; // Vacuum pumps started while venting was active
    E4501_TemperatureDroppedBelow280K             : UDINT := 4500002; // One or more temperatures dropped below 280 K during venting
    E4502_LN2RefillingStartedDuringVenting        : UDINT := 4500003; // LN2 refilling became active during venting
    E4503_RegenerationStartedDuringVenting        : UDINT := 4500004; // Sorption pump regeneration became active during venting
    E4504_GN2HoseDisconnectedDuringVenting        : UDINT := 4500005; // GN2 hose was disconnected during venting

    // --- [4600] Shutdown / Recovery Failures ---
    E4600_VentingValvesDidNotClose                : UDINT := 4600001; // Venting valves failed to close during stop
    E4601_VentingShutdownTimeout                  : UDINT := 4600002; // Venting shutdown did not complete in time
    E4602_SystemNotAtSafePressureAfterVenting     : UDINT := 4600003; // System not at safe pressure after venting completed

END_VAR


M_Configure();

M_ReadSensors();

M_HandleEvents();

M_ExecuteControllers();

M_UpdateStatus();

M_StateMachine(interlocks := interlocks);



IF bReset_Valves THEN
	M_ResetValves();
	bReset_Valves := FALSE;
END_IF

METHOD M_Activity_Check_Preconditions
VAR_INPUT
END_VAR

// CHECK_Venting_PRECONDITIONS

stat.bActive := TRUE;
stat.bBusy := FALSE; 
stat.bDone := FALSE;  

// --- Precondition Check: Venting Valves Closed ---
IF NOT in_Cryo_Stat.bVentingValvesAreClosed THEN
    stat.nState := E_MET_CRYO_VENTING_STATE.ERROR;
    stat.sState := 'Error: Venting valves are not closed.';
    RETURN; 
END_IF

// --- Precondition Check: Pumps Running ---
IF in_Cryo_Stat.bPumpsAreRunning THEN
    stat.nState := E_MET_CRYO_VENTING_STATE.ERROR;
    stat.sState := 'Error: Pumps are running.';
    RETURN; 
END_IF

// --- Precondition Check: Evacuation Stopped ---
IF in_Cryo_Stat.bEvacuationActive THEN
    stat.nState := E_MET_CRYO_VENTING_STATE.ERROR;
    stat.sState := 'Error: Evacuation Active.';
    RETURN; 
END_IF

// --- Precondition Check: Cool Down Active ---
IF in_Cryo_Stat.bCoolDownActive THEN
    stat.nState := E_MET_CRYO_VENTING_STATE.ERROR;
    stat.sState := 'Error: Cool down is active.';
    RETURN; 
END_IF

// --- Precondition Check: Cool Down Active ---
IF in_Cryo_Stat.bRegenerationActive THEN
    stat.nState := E_MET_CRYO_VENTING_STATE.ERROR;
    stat.sState := 'Error: Regeneration is active.';
    RETURN; 
END_IF

// --- Precondition Check: Cool Down Active ---
IF NOT in_Cryo_Stat.bGN2SupplyConnected THEN
    stat.nState := E_MET_CRYO_VENTING_STATE.ERROR;
    stat.sState := 'Error: GN2 supply not connected.';
    RETURN; 
END_IF

IF in_Cryo_Stat.lrLowestTempK < 280 THEN
    stat.nState := E_MET_CRYO_VENTING_STATE.ERROR;
    stat.sState := 'Error: All temperatures are NOT above 280K.';
    RETURN;
END_IF


stat.nState := E_MET_CRYO_VENTING_STATE.PREPARE_FOR_VENTING;
stat.sState := 'Preconditions met. Waiting for the timeout..';
END_METHOD

METHOD M_Activity_ClosingValve
VAR_INPUT
	index:		INT;
	nNextState:	E_CRYO_EVAC_STATE_50000;	// Next state after valve is closed
END_VAR
//// Check if valve index is valid.
//// If not, just return (for safety).
//IF index < 1  OR  index > 2	THEN
//	RETURN;
//END_IF 

//IF ptrV[index]^.stat.bActOFF THEN
//	// The valve is closed.
//	// Set next state and execute its action
//	M_SetNextState(nNextState);	// Next state
	
//END_IF
END_METHOD

METHOD M_Activity_Error_Handling
VAR_INPUT
END_VAR
VAR_IN_OUT
	interlocks:						T_METIS_CRYO_INTERLOCKS;
END_VAR
stat.bError := TRUE;

M_Close_Venting_Valves();

IF ctrl.bReset THEN
	M_ResetValves(); 
	stat.nState := E_MET_CRYO_VENTING_STATE.NONE;
	ctrl.bReset := FALSE;
	ctrl.bEnable := FALSE;						
END_IF
END_METHOD

METHOD M_Activity_None
VAR_INPUT
END_VAR
VAR_IN_OUT
	{attribute 'OPC.UA.DA' := '0'}
	interlocks:						T_METIS_CRYO_INTERLOCKS;
END_VAR
stat.bActive := FALSE;
stat.bError := FALSE;
M_Close_Venting_Valves();

// Check enable AND Interlocks
IF trigEnable.Q AND NOT interlocks.bInterlock_Venting THEN
	stat.nState := E_MET_CRYO_VENTING_STATE.CHECK_PRECONDITIONS;
	logs.M_LogInfo('VENTING started by the operator.');
ELSE
	stat.nState := E_MET_CRYO_VENTING_STATE.NONE;
	stat.sState := 'Venting OFF';
END_IF
END_METHOD

METHOD M_Activity_OpeningValve
VAR_INPUT
	index:		INT;
	nNextState:	E_CRYO_EVAC_STATE_50000;	// Next state after valve is closed
END_VAR
//IF NOT in_bEnable THEN
//	// If system is disabled, start stopping procedure.
//	M_SetNextState(E_CRYO_EVAC_STATE_50000.CLOSE_ALL_VALVES);	// Next state
	
//ELSIF ptrV[index]^.stat.bActON THEN
//	// The valve is open.
//	// Go to next state
//	M_SetNextState(nNextState);
	
//END_IF
END_METHOD

METHOD M_Activity_Prepare_For_Venting
VAR_INPUT
END_VAR
VAR

    
END_VAR
VAR_INST
	bTimerActive         : BOOL := FALSE; // Ensures timer starts only once
	fbWaitTimer          : TON;
    trigStartTimer       : R_TRIG;
END_VAR


IF NOT bTimerActive THEN
    fbWaitTimer(IN := TRUE, PT := cfg.tWaitingTimeToStartVenting);
    bTimerActive := TRUE;
    stat.sState := 'Waiting before starting Venting...';
END_IF



fbWaitTimer(IN := NOT trigDisable.Q); // Cancel timer if operator cancels

IF trigDisable.Q THEN
	stat.sState := 'Venting cancelled by operator';
	stat.nState := E_MET_CRYO_VENTING_STATE.FINISHED;
	fbWaitTimer(IN := FALSE);
	bTimerActive := FALSE;

ELSIF fbWaitTimer.Q THEN
	stat.sState := 'Timeout complete. Starting Venting...';
	stat.nState := E_MET_CRYO_VENTING_STATE.START_VENTING;
	fbWaitTimer(IN := FALSE);
	bTimerActive := FALSE;
ELSE
	stat.nState := E_MET_CRYO_VENTING_STATE.PREPARE_FOR_VENTING;
	stat.sState := CONCAT('Waiting for timeout or operator action...',
							 F_TON_TO_TIME_STRING(Timer := fbWaitTimer));
END_IF
END_METHOD

METHOD M_Activity_Start_Venting
VAR_INPUT
END_VAR
//VAR_INST
//	i: INT := 0;
//END_VAR
VAR
    Timeout           : TON := (PT := T#5s);   // 5-second timeout
    bStartAttempted     : BOOL := FALSE;
END_VAR

M_HandleInterlocks();
IF stat.bError THEN
    stat.sState := 'Interlocks not satisfied – aborting start';
    stat.nState := E_MET_CRYO_VENTING_STATE.ERROR;
    stat.bBusy  := FALSE;
    RETURN;
END_IF


stat.bActive := TRUE;
stat.bBusy := TRUE;
stat.bDone := FALSE;

//// Venting valves opening sequence
//IF NOT bStartAttempted THEN
//    stat.sState := 'Opening Venting Valves...';
    M_Open_Venting_Valves();
//    Timeout(IN := TRUE);
//    bStartAttempted := TRUE;
//    RETURN;    
//END_IF

//// Check valve status
//IF NOT in_Cryo_Stat.bVentingValvesAreClosed THEN
//    Timeout(IN := FALSE);  
//    stat.sState := 'Venting in progress';
    stat.nState := E_MET_CRYO_VENTING_STATE.VENTING_IN_PROGRESS;
//    stat.bBusy := TRUE;
//    stat.bDone := TRUE;
//ELSIF Timeout.Q THEN
//    stat.sState := 'Error: Venting Valves failed to open';
//    stat.nState := E_MET_CRYO_VENTING_STATE.ERROR;
//    stat.bBusy := FALSE;
//    Timeout(IN := FALSE);
//END_IF
END_METHOD

METHOD M_Activity_Stop_Venting
VAR_INPUT
END_VAR
//VAR_INST
//	i : INT := 0;
//END_VAR
VAR
    nRetries        : INT := 0;
    fbTimeout       : TON := (PT := T#5s);
    bClosingStarted : BOOL := FALSE;
END_VAR

IF NOT bClosingStarted THEN
    M_Close_Venting_Valves();
    bClosingStarted := TRUE;
    fbTimeout(IN := TRUE);
END_IF

IF NOT in_Cryo_Stat.bVentingValvesAreClosed THEN
    IF fbTimeout.Q THEN
        stat.sState := 'Venting Valves failed to Close';
        stat.nState := E_MET_CRYO_VENTING_STATE.ERROR;
    ELSE
        IF nRetries < 3 THEN
            M_Close_Venting_Valves(); // Retry attempt
            nRetries := nRetries + 1;
        END_IF
    END_IF
ELSE
    fbTimeout(IN := FALSE);
    stat.sState := 'Venting Valves Closed';
    stat.nState := E_MET_CRYO_VENTING_STATE.FINISHED;
END_IF

//stat.sState := 'Stopping Venting...';

//M_Close_Venting_Valves();

//IF NOT in_Cryo_Stat.bVentingValvesAreClosed THEN
//	IF i >= 10 THEN
//		IF in_Cryo_Stat.bVentingValvesAreClosed THEN
//			stat.nState := E_MET_CRYO_VENTING_STATE.FINISHED;
//		ELSE
//			stat.sState := 'Venting Valves failed to Close';
//			stat.nState := E_MET_CRYO_VENTING_STATE.ERROR;
//		END_IF
//	END_IF
//	i := i + 1;
//ELSE
//	stat.nState := E_MET_CRYO_VENTING_STATE.FINISHED;
//END_IF
END_METHOD

METHOD M_Activity_Venting_InProgress
VAR_INPUT
END_VAR

M_HandleInterlocks();

// IF Venting is not stopped manually 

IF NOT trigDisable.Q THEN 
	
	// Check if HPG pressre is valid and greater than cfg.trigVentingPressureAchieved
	
//	IF HPG.stat.bValid AND (HPG.tat.lrPressure >= cfg.lrMaxVentingPressure) THEN

	IF HPG.stat.bValid AND (HPG.stat.lrPressure >= (in_Cryo_Stat.lrAmbientPressure + 50)) THEN
			stat.nState := E_MET_CRYO_VENTING_STATE.STOPPING_VENTING;
			stat.sState := 'Venting Finished';
			logs.M_LogInfo('Pressure achieved. VENTING stopped automatically.');
			
	ELSE
			(*TODO once the pressure vote or guages have get ramp feature*)
			// Check if pressure is increasing positively	
			//sensor_HPG1.
	
			stat.nState := E_MET_CRYO_VENTING_STATE.VENTING_IN_PROGRESS;
			stat.sState := 'Venting...';
	END_IF

ELSE
	stat.nState := E_MET_CRYO_VENTING_STATE.STOPPING_VENTING;
	stat.sState := 'Venting Stopped Manually';
	logs.M_LogInfo('VENTING stopped by the operator.');
END_IF
END_METHOD

METHOD M_AreVentingValvesClosed : BOOL
VAR_INPUT
END_VAR

IF N2V_1.stat.bActON OR N2V_2.stat.bActON THEN
	M_AreVentingValvesClosed := FALSE;
ELSE
	M_AreVentingValvesClosed := TRUE; 
END_IF
END_METHOD

METHOD M_Close_Venting_Valves
VAR_INPUT
END_VAR

// Close venting valves

ctrl.bEnable_N2V_1 := FALSE;
ctrl.bEnable_N2V_2 := FALSE;
END_METHOD

METHOD M_Configure
VAR_INPUT
END_VAR





//ctrl.bEnable_N2V_1 := in_bEnable_N2V_1;
//ctrl.bEnable_N2V_2 := in_bEnable_N2V_2;

IF NOT bConfigured THEN
	
	// Set pointers to Valves - MUST!!!
	ptrV[1]	:= ADR(N2V_1);
	ptrV[2]	:= ADR(N2V_2);
	
	
	// Set pointers to Valve Commands - MUST!!!
	ptrVC[1]	:= ADR(ctrl.cor_N2V_1);
	ptrVC[2]	:= ADR(ctrl.cor_N2V_2);
	
	
	// Set pointers to Enable Valves flags - MUST!!!
	ptrEV[1]	:= ADR(ctrl.bEnable_N2V_1);
	ptrEV[2]	:= ADR(ctrl.bEnable_N2V_2);
	
	
	// Enable power of the pressure sensors

	bPwr_HPG1	:= TRUE;		
	bPwr_HPG2	:= TRUE;

	M_ResetValves();		
	
	// This call just configures logs at the very start.
	// Logging is done by explicit calls to M_LogInfo().
	logs(in_sName := in_sName);	
	
	bConfigured := TRUE;

END_IF
END_METHOD

METHOD M_ExecuteControllers
VAR_INPUT
END_VAR
// Valve commands
ctrl.cor_N2V_1(in_bEnable := ctrl.bEnable_N2V_1);	// Handling of PVV1 commands
ctrl.cor_N2V_2(in_bEnable := ctrl.bEnable_N2V_2);	// Handling of PVV2 commands


// Valve Control

IF N2V_1.stat.bError THEN
	N2V_1.M_Reset();
END_IF

N2V_1(
	in_bEnable			:= ctrl.cor_N2V_1.out_bEnable,
	in_nFeedback		:= E_CRYO_BIN_ACT_FEEDBACK.ON_ONLY);

IF N2V_2.stat.bError THEN
	N2V_2.M_Reset();
END_IF
	
N2V_2(
	in_bEnable			:= ctrl.cor_N2V_2.out_bEnable,
	in_nFeedback		:= E_CRYO_BIN_ACT_FEEDBACK.ON_ONLY);
END_METHOD

METHOD M_HandleEvents
VAR_INPUT
END_VAR

//
// Handle triggers
//

trigEnable	(CLK := ctrl.bEnable);
trigDisable	(CLK := ctrl.bEnable);
END_METHOD

METHOD M_HandleInterlocks
VAR_INPUT
END_VAR


// Venting Valves Closed ---
IF in_Cryo_Stat.bVentingValvesAreClosed THEN
    stat.nState := E_MET_CRYO_VENTING_STATE.ERROR;
    stat.sState := 'Error: Venting valves are closed.';
    RETURN; 
END_IF

// Pumps Running ---
IF in_Cryo_Stat.bPumpsAreRunning THEN
    stat.nState := E_MET_CRYO_VENTING_STATE.ERROR;
    stat.sState := 'Error: Pumps are Running.';
    RETURN; 
END_IF

// --- Evacuation Activated ---
IF in_Cryo_Stat.bEvacuationActive THEN
    stat.nState := E_MET_CRYO_VENTING_STATE.ERROR;
    stat.sState := 'Error: Evacuation Activated.';
    RETURN; 
END_IF

// --- Cool Down Active ---
IF in_Cryo_Stat.bCoolDownActive THEN
    stat.nState := E_MET_CRYO_VENTING_STATE.ERROR;
    stat.sState := 'Error: Cool down activated.';
    RETURN; 
END_IF

// --- Regeneration Active ---
IF in_Cryo_Stat.bRegenerationActive THEN
    stat.nState := E_MET_CRYO_VENTING_STATE.ERROR;
    stat.sState := 'Error: Regeneration activated.';
    RETURN; 
END_IF

// --- GN2 supply disconnected ---
IF NOT in_Cryo_Stat.bGN2SupplyConnected THEN
    stat.nState := E_MET_CRYO_VENTING_STATE.ERROR;
    stat.sState := 'Error: GN2 supply  disconnected.';
    RETURN; 
END_IF

IF HPG.stat.lrPressure > (in_Cryo_Stat.lrAmbientPressure + 10) THEN
    stat.nState := E_MET_CRYO_VENTING_STATE.ERROR;
    stat.sState := 'Error: Pressure in vessle too high';
	(*TODO: Implement critical Alarm*)
    RETURN;
END_IF
END_METHOD

METHOD M_IsVentingFinishedSuccessfully : BOOL
VAR_INPUT
END_VAR

IF stat.nState = E_MET_CRYO_VENTING_STATE.FINISHED THEN
	M_IsVentingFinishedSuccessfully := stat.bVentingPressureAchieved;	
END_IF
END_METHOD

METHOD M_Open_Venting_Valves
VAR_INPUT
END_VAR


// Open venting valves

ctrl.bEnable_N2V_1 := TRUE;
ctrl.bEnable_N2V_2 := TRUE;
END_METHOD

METHOD M_ReadSensors
VAR_INPUT
END_VAR


sensor_HPG1(in_sName:= 'HPG1_Sen', in_nType:= E_CRYO_SENSOR_TYPE_PRESS.CMR_361, in_nSampleTime:= 100);
sensor_HPG2(in_sName:= 'HPG2_Sen', in_nType:= E_CRYO_SENSOR_TYPE_PRESS.CMR_361, in_nSampleTime:= 100);


ctrl.por_HPG(in_bEnable := ctrl.bSim_Press_HPG);	// Simulation flag override
HPG(
	in_sName:= 'HPG', 
	in_bSimulation:= ctrl.por_HPG.out_bEnable, 
	in_nNumSensor:= 2, 
	in_nVoteMethod:= , 
	in_pSensor1:= ADR(sensor_HPG1), 
	in_pSensor2:= ADR(sensor_HPG2));
	
ctrl.por_HPG1(in_bEnable := ctrl.bSim_Press_HPG1);	// Simulation flag override	
HPG1(
	in_sName:= 'HPG1', 
	in_bSimulation:= ctrl.por_HPG1.out_bEnable, 
	in_nNumSensor:= 1, 
	in_nVoteMethod:= , 
	in_pSensor1:= ADR(sensor_HPG1), 
	in_pSensor2:= , 
	in_pSensor3:= , 
	in_pSensor4:= , 
	in_pSensor5:= );

ctrl.por_HPG2(in_bEnable := ctrl.bSim_Press_HPG2);	// Simulation flag override		
HPG2(
	in_sName:= 'HPG2', 
	in_bSimulation:= ctrl.por_HPG2.out_bEnable, 
	in_nNumSensor:= 1, 
	in_nVoteMethod:= , 
	in_pSensor1:= ADR(sensor_HPG2), 
	in_pSensor2:= , 
	in_pSensor3:= , 
	in_pSensor4:= , 
	in_pSensor5:= );
END_METHOD

METHOD M_ResetValves
VAR_INPUT
END_VAR
N2V_1.M_Reset();
N2V_2.M_Reset();
END_METHOD

METHOD PRIVATE M_SetError
VAR_INPUT
    nCode     : UDINT;
    sMessage  : STRING;
END_VAR


stat.Error.nCode := nCode;
stat.Error.sMessage := sMessage;
stat.bError := TRUE;
stat.nState := E_MET_CRYO_VENTING_STATE.ERROR;
END_METHOD

METHOD M_StateMachine
VAR_INPUT
END_VAR
VAR_IN_OUT
	{attribute 'OPC.UA.DA' := '0'}
	interlocks:						T_METIS_CRYO_INTERLOCKS;
END_VAR

//--- State Machine Logic ---
CASE stat.nState OF
	
	E_MET_CRYO_VENTING_STATE.NONE:
	
		M_Activity_None(interlocks := interlocks);
	
	E_MET_CRYO_VENTING_STATE.CHECK_PRECONDITIONS:
		
		M_Activity_Check_Preconditions();
		
	E_MET_CRYO_VENTING_STATE.PREPARE_FOR_VENTING:
	
		M_Activity_Prepare_For_Venting();
		
	E_MET_CRYO_VENTING_STATE.START_VENTING:
	
		M_Activity_Start_Venting();
	
	E_MET_CRYO_VENTING_STATE.VENTING_IN_PROGRESS:
		
		M_Activity_Venting_InProgress();
		
	E_MET_CRYO_VENTING_STATE.STOPPING_VENTING:
	
		M_Activity_Stop_Venting();	
	
	E_MET_CRYO_VENTING_STATE.FINISHED:
	
			stat.sState := 'Venting Finished';
			stat.nState := E_MET_CRYO_VENTING_STATE.NONE;
			ctrl.bEnable := FALSE;		
			stat.bActive := FALSE;
			stat.bBusy := FALSE; 
			stat.bDone := TRUE;

	E_MET_CRYO_VENTING_STATE.ERROR:
		M_Activity_Error_Handling(interlocks := interlocks);


END_CASE
END_METHOD

METHOD M_UpdateStatus
VAR_INPUT
END_VAR
VAR
	m_bVentingPressureAchieved: BOOL;
END_VAR
stat.bEnabled		:= ctrl.bEnable;

// References are set once the evacuation system is configured.
IF stat.bConfigured	THEN
	//stat.bRootPumpON	:= rpRef.M_IsReady();
	//stat.bTurboPumpON	:= tpRef.M_IsReady();
END_IF

out_bVentingActive := stat.bActive;

m_bVentingPressureAchieved := (HPG.stat.lrPressure >= in_Cryo_Stat.lrAmbientPressure);

stat.bVentingPressureAchieved := m_bVentingPressureAchieved; 

trigVentingPressureAchieved (CLK := m_bVentingPressureAchieved);


// Check Pre-Conditions for HMI Enable 


stat.bPreConditionsMet := 	NOT in_Cryo_Stat.bPumpsAreRunning 	 AND
							NOT in_Cryo_Stat.bEvacuationActive   AND
							NOT in_Cryo_Stat.bCoolDownActive     AND
							NOT in_Cryo_Stat.bRegenerationActive AND
							in_Cryo_Stat.bGN2SupplyConnected 	 AND
							in_Cryo_Stat.lrLowestTempK > 280.0;
END_METHOD

END_FUNCTION_BLOCK

// POUs/Functions/F_TON_TO_TIME_STRING
// Returns the remaining time
FUNCTION F_TON_TO_TIME_STRING : STRING[50]
VAR_INPUT
    Timer : TON;   // TON instance
END_VAR
VAR_OUTPUT
    sElapsed   : STRING[50];  // "HH:MM:SS elapsed"

END_VAR
VAR
	sRemaining : STRING[50];  // "HH:MM:SS remaining"
    tElapsed, tRemaining : TIME;
    iEH, iEM, iES        : DINT;   // elapsed H:M:S
    iRH, iRM, iRS        : DINT;   // remaining H:M:S
    lrSec                : LREAL;
    sEH, sEM, sES        : STRING[3];
    sRH, sRM, sRS        : STRING[3];
END_VAR

// --- Elapsed time ---
tElapsed := Timer.ET;
lrSec := TIME_TO_LREAL(tElapsed) / 1000.0;   // TIME is ms
iEH := TRUNC(lrSec / 3600.0);
iEM := TRUNC((lrSec - iEH * 3600) / 60.0);
iES := TRUNC(lrSec - iEH * 3600 - iEM * 60);

// Pad with zeros
IF iEH < 10 THEN sEH := CONCAT('0', DINT_TO_STRING(iEH)); ELSE sEH := DINT_TO_STRING(iEH); END_IF;
IF iEM < 10 THEN sEM := CONCAT('0', DINT_TO_STRING(iEM)); ELSE sEM := DINT_TO_STRING(iEM); END_IF;
IF iES < 10 THEN sES := CONCAT('0', DINT_TO_STRING(iES)); ELSE sES := DINT_TO_STRING(iES); END_IF;

sElapsed := CONCAT(CONCAT(CONCAT(sEH, ':'), CONCAT(sEM, ':')), sES);
sElapsed := CONCAT(sElapsed, ' elapsed');

// --- Remaining time ---
tRemaining := Timer.PT - Timer.ET;
IF tRemaining < T#0s THEN
    tRemaining := T#0s;  // Clamp at zero
END_IF;

lrSec := TIME_TO_LREAL(tRemaining) / 1000.0;
iRH := TRUNC(lrSec / 3600.0);
iRM := TRUNC((lrSec - iRH * 3600) / 60.0);
iRS := TRUNC(lrSec - iRH * 3600 - iRM * 60);

// Pad with zeros
IF iRH < 10 THEN sRH := CONCAT('0', DINT_TO_STRING(iRH)); ELSE sRH := DINT_TO_STRING(iRH); END_IF;
IF iRM < 10 THEN sRM := CONCAT('0', DINT_TO_STRING(iRM)); ELSE sRM := DINT_TO_STRING(iRM); END_IF;
IF iRS < 10 THEN sRS := CONCAT('0', DINT_TO_STRING(iRS)); ELSE sRS := DINT_TO_STRING(iRS); END_IF;

sRemaining := CONCAT(CONCAT(CONCAT(sRH, ':'), CONCAT(sRM, ':')), sRS);
sRemaining := CONCAT(sRemaining, ' remaining');

// Returns the remaining time
F_TON_TO_TIME_STRING := sRemaining;

END_FUNCTION

// POUs/Routines/CoolDown/FB_METIS_CRYO_COOL_DOWN
FUNCTION_BLOCK FB_METIS_CRYO_COOL_DOWN
VAR_INPUT
	in_sName:							STRING := 'COOL-DOWN';
	in_Cryo_Stat:							T_METIS_CRYO_STAT;
	in_RefVAGF:					REFERENCE TO FB_CRYO_PRESSURE_VOTE;
	in_RefVAGG:					REFERENCE TO FB_CRYO_PRESSURE_VOTE;
	
		// System commands for Valve1 and Valve2
	in_bEnable_PVV_P1:					BOOL:= FALSE;
	in_bEnable_PVV_P2:					BOOL:= FALSE;
	in_bEnable_PVV_P3:					BOOL:= FALSE;
	
	in_lrCoolDown_PreCond_Press: 		LREAL := 0.0001; // p<1e-4 mbar pressure
	in_lrLN2_TempK:						LREAL; 	 // LN2 detection temp threshold
	in_lrRadShld_TempK_TO_Start_PTCs:	LREAL; 	 // LN2 detection temp threshold
	
END_VAR
VAR_OUTPUT
	out_bCoolDownActive:		BOOL := FALSE;
END_VAR
VAR_IN_OUT
	{attribute 'OPC.UA.DA' := '0'}
	all_cryo_temps:					FB_METIS_TEMPERATURES;
	{attribute 'OPC.UA.DA' := '0'}
	all_heaters:					FB_METIS_HEATERS;
	{attribute 'OPC.UA.DA' := '0'}
	all_t_ctrls:      				FB_METIS_TCTRL;
	{attribute 'OPC.UA.DA' := '0'}
	all_t_votes: 					FB_METIS_VOTERS;
	{attribute 'OPC.UA.DA' := '0'}
	interlocks:						T_METIS_CRYO_INTERLOCKS;
END_VAR
VAR
		/////////////////////
	// Cryo System logs
	/////////////////////
		
	logs:	FB_CRYO_FUNCTION_LOG;
	////////////////////////
	// Pre-Cooling valves//
	//////////////////////
	PVV_P1:		FB_CRYO_VALVE_CTRL;		// Pre-Cooling valve 1
	PVV_P2:		FB_CRYO_VALVE_CTRL;		// Pre-Cooling valve 2
	PVV_P3:		FB_CRYO_VALVE_CTRL;		// Pre-Cooling valve 3
	
	
	// Pointers to valves
	ptrV:	ARRAY [1..3] OF POINTER TO FB_CRYO_VALVE_CTRL;
	// Pointers to valve commands
	ptrVC:	ARRAY [1..3] OF POINTER TO FB_CRYO_CMD_OVERRIDE;
	// Pointers to Enable flags for valves
	ptrEV:	ARRAY [1..3] OF POINTER TO BOOL;
	
	
	
	cmdPVV_P1:	FB_CRYO_ACTUATOR_CMD;	// Handling of PVV_P1 command
	cmdPVV_P2:	FB_CRYO_ACTUATOR_CMD;	// Handling of PVV_P2 command
	cmdPVV_P3:	FB_CRYO_ACTUATOR_CMD;	// Handling of PVV_P3 command
	
	///////////////////////
	// LN2 Level Control//
	//////////////////////
	{attribute 'TcHmiSymbol.Show'}
	lc_ln2_level_ctrl: ARRAY [1..3] OF FB_METIS_CRYO_LN2_LEVEL_CTRL; // Automatic LN2 filling based on LN2 level

	// Indexes for Engineering GUIs.
	gui_index_ln2_ctrl:			INT := 1;
	
	// For ESO Framework to read them to display on Grafana
	{attribute 'OPC.UA.DA' := '1'}
	lrLN2_Level_Sensor_1_HA_TempK:		LREAL;
	{attribute 'OPC.UA.DA' := '1'}
	lrLN2_Level_Sensor_1_H_TempK:		LREAL;
	{attribute 'OPC.UA.DA' := '1'}
	lrLN2_Level_Sensor_1_L_TempK:		LREAL;
	{attribute 'OPC.UA.DA' := '1'}
	lrLN2_Level_Sensor_1_LA_TempK:		LREAL;
	{attribute 'OPC.UA.DA' := '1'}
	lrLN2_Level_Sensor_2_HA_TempK:		LREAL;
	{attribute 'OPC.UA.DA' := '1'}
	lrLN2_Level_Sensor_2_H_TempK:		LREAL;
	{attribute 'OPC.UA.DA' := '1'}
	lrLN2_Level_Sensor_2_L_TempK:		LREAL;
	{attribute 'OPC.UA.DA' := '1'}
	lrLN2_Level_Sensor_2_LA_TempK:		LREAL;
	{attribute 'OPC.UA.DA' := '1'}
	lrLN2_Level_Sensor_3_HA_TempK:		LREAL;
	{attribute 'OPC.UA.DA' := '1'}
	lrLN2_Level_Sensor_3_H_TempK:		LREAL;
	{attribute 'OPC.UA.DA' := '1'}
	lrLN2_Level_Sensor_3_L_TempK:		LREAL;
	{attribute 'OPC.UA.DA' := '1'}
	lrLN2_Level_Sensor_3_LA_TempK:		LREAL;
	
	
	////////////
	// Pressure
	////////////
	
	// Pressure transducers
	sensor_VAG_PCA:	FB_CRYO_SENSOR_PRESSURE;	// Cooling circuit pressure gauge #1
	sensor_VAG_PCB:	FB_CRYO_SENSOR_PRESSURE;	// Cooling circuit pressure gauge #2
	sensor_VAG_P1:	FB_CRYO_SENSOR_PRESSURE;	// Cooling circuit pressure gauge #3

	{attribute 'TcHmiSymbol.Show'}
	VAG_PCA:	FB_CRYO_PRESSURE_VOTE;			// Precooling pressure
	{attribute 'TcHmiSymbol.Show'}	
	VAG_PCB:	FB_CRYO_PRESSURE_VOTE;			// Precooling pressure
	{attribute 'TcHmiSymbol.Show'}
	VAG_P1:	FB_CRYO_PRESSURE_VOTE;				// Precooling pressure
	
	// Pressure sensors IDN resistors
	
	nIdnRes_VAG_PCA		AT %I* :INT;
	nIdnRes_VAG_PCB		AT %I* :INT;
	nIdnRes_VAG_P1		AT %I* :INT;
	
	// Pressure sensor power 24V Dig Out
	
	bPwr_VAG_PCA		AT %Q* :BOOL;
	bPwr_VAG_PCB        AT %Q* :BOOL;
	bPwr_VAG_P1         AT %Q* :BOOL;

	
//	// Pressure measurements
//	VAG1:	FB_CRYO_PRESSURE_VOTE;				// Prevacuum pressure #1
//	VAG2:	FB_CRYO_PRESSURE_VOTE;				// Prevacuum pressure #2
//	VAG3:	FB_CRYO_PRESSURE_VOTE;				// Prevacuum pressure #3
//	// VAGF and VAGG are just copies of in_RefVAGF and in_RefVAGG !!!
//	VAGF:	FB_CRYO_PRESSURE_VOTE;				// Cryo pressure F
//	VAGG:	FB_CRYO_PRESSURE_VOTE;				// Cryo pressure G

//	// Pointers to pressures
//	ptrP:	ARRAY [1..5] OF POINTER TO FB_CRYO_PRESSURE_VOTE;
	
		
	
	cfg:	T_MET_CRYO_COOLDOWN_CFG;
	ctrl:	T_MET_CRYO_COOLDOWN_CTRL;
	stat:	T_MET_CRYO_COOLDOWN_STAT;
	
	
	timer:	TON;
	trig:	R_TRIG;	// Start trigger
	
	// GUI stuff
	guiValveIndex:	UINT := 1;	// Index for Valve Engineering GUI
	
	
	// Configure
	bConfigured:		BOOL := FALSE;
	
	
	bReset_Valves:		BOOL:= FALSE;
	
	///////////////////////
	///// PTC Coolers /////
	//////////////////////	
	
	// Compressors for Pulse-Tube Cooler
	
	ptc:				ARRAY [1..3] OF FB_METIS_CRYO_CPA;
		
	// Pointers to System Overrides for control and sensors.
	// See M_Configure() for pointer assignments.
	//
	// Pointers to Overrides of Enable commands for valves, pumps and coolers.
	ptrArr_cor_ptcs:	ARRAY [1..3] OF POINTER TO FB_CRYO_CMD_OVERRIDE;
	//
	// Indexes for Override GUIs.
	//
	guiIndex_cor_ptcs:	UINT := 1;	// Index for Command Override Engineering GUI
	
	////////////////////////////////
	///// LN2 Supply from ESO /////
	//////////////////////////////
	
	bESO_LN2_Supply AT %I*: BOOL;
	
	bSimulated_ESO_Supply_Flag AT %Q*: BOOL := TRUE;
	
	
	// Simulated temp for level sensors
	nSim_LN2_LS_TempK:	ARRAY [1..12] OF INT := 
	[105, 105, 105, 84, 105, 105, 105, 84,105, 105, 105, 84];
	
	nSim_Temp_HA_1	AT %Q*	:		INT;
	nSim_Temp_H_1	AT %Q*	:		INT;
	nSim_Temp_L_1	AT %Q*	:		INT;
	nSim_Temp_LA_1	AT %Q*	:		INT;
	
	nSim_Temp_HA_2	AT %Q*	:		INT;
	nSim_Temp_H_2	AT %Q*	:		INT;
	nSim_Temp_L_2	AT %Q*	:		INT;
	nSim_Temp_LA_2	AT %Q*	:		INT;
	
	nSim_Temp_HA_3	AT %Q*	:		INT;
	nSim_Temp_H_3	AT %Q*	:		INT;
	nSim_Temp_L_3	AT %Q*	:		INT;
	nSim_Temp_LA_3	AT %Q*	:		INT;
	
	nSim_Status		AT %Q*	:   UINT;
	nSimCouplerState AT %Q*	:   INT := 8;
	/////////////
	// Timers //
	///////////
	
	tDelay_SHB:		TON;
	tDelay_SHC:		TON;
	
	tDelay_SHs_Cold:		TON;
	
	tDelaySHB:			TIME; // := T#900S;
	tDelaySHC:			TIME; // := T#900S;
	tDelaySHCold:		TIME; // := T#4H;
	
	lrDelaySHB:			LREAL := 900.0;
	lrDelaySHC:			LREAL := 900.0;
	lrDelaySHCold:		LREAL := 4.0;
	
	tDelayPTC_1:	TON;
	tDelayPTC_2:	TON;
	tDelayPTC_3:	TON;
	
	tDelayPTCStart: TIME := T#30S;
	
	bAllowPTCsStart:	BOOL := FALSE;
	
	// Triggers.
	//
	// Capture Enable/Disable.
	trigEnable:		R_TRIG;	// in_bEnable
	trigDisable:	F_TRIG;	// in_bEnable
	
	(****************************
	***** Early Refilling *******
	****************************)
	
    // Latches: each vessel has reached HIGH at least once
    bHighReachedSHA : BOOL := FALSE;   // lc_ln2_level_ctrl[1]
    bHighReachedSHB : BOOL := FALSE;   // lc_ln2_level_ctrl[2]
    bHighReachedSHC : BOOL := FALSE;   // lc_ln2_level_ctrl[3]

    // Overall early refilling active flag
    bEarlyRefillingActive : BOOL := FALSE;
	bEarlyRefillDone:		BOOL := TRUE; // Start with done, so we canr restart again

    // Timers
    tonEarlyRefillTotal  : TON;        // 24 h total early refilling time
    tonEarlyRefillCycle  : TON;        // 2 h cycle between refills

    // Configurable times
    tEarlyRefillTotal    : TIME; // := T#24H;
    tEarlyRefillCycle    : TIME; // := T#2H;
	
	lrEarlyRefillTotal:		LREAL := 24.0;
	lrEarlyRefillCycle:		LREAL := 2.0;

    // Helper to restart the 2 h cycle timer cleanly
    bRestartCycle        : BOOL := FALSE;
	
	// StandAlone Filling if we restart in a cold shield state
	bStandaloneLN2Filling: 		BOOL := FALSE; 

END_VAR
VAR CONSTANT

    // --- [1000] Preconditions ---
    E1000_PressureTooHigh                         : UDINT := 1000001; // System pressure > 1e-4 mbar
    E1001_WarmUpHeatersActive                     : UDINT := 1000002; // Warm-up heaters are active
    E1002_SorptionHeaterActive                    : UDINT := 1000003; // Sorption heater is active
    E1003_VentingValveOpen                        : UDINT := 1000004; // Venting valve is not closed
    E1004_PumpsNotRunning                         : UDINT := 1000005; // Vacuum pumps not running or TMP not at speed
    E1005_LN2SupplyNotReady                       : UDINT := 1000006; // LN2 supply not ready
	E1006_EvacuationNotActive                     : UDINT := 1000007; // LN2 supply not ready

    // --- [1100] Valve Operation Errors ---
    E1100_SHA_V_Error	                          : UDINT := 1100001; // Valve SHA.V failed to open in time
    E1101_SHB_V_Error   	                      : UDINT := 1100002; // Valve SHB.V failed to open in time
    E1102_SHC_V_Error							  : UDINT := 1100003; // Valve SHC.V failed to open in time
    E1103_PCB_C1_FailedToOpen                     : UDINT := 1100004; // PCB.C1 did not reach 50% after command
    E1104_PCB_C2_FailedToOpen                     : UDINT := 1100005; // PCB.C2 did not open
    E1105_PCA_C1_FailedToOpen                     : UDINT := 1100006; // PCA.C1 did not reach 50% after command
    E1106_PCA_C2_FailedToOpen                     : UDINT := 1100007; // PCA.C2 did not open
    E1107_PCB_VV_FailedToOpenOrClose              : UDINT := 1100008; // PCB.VV failed operation
    E1108_PCA_VV_FailedToOpenOrClose              : UDINT := 1100009; // PCA.VV failed operation
    E1109_PVV_SwitchingConflict                   : UDINT := 1100010; // PVV valves not in correct configuration

    // --- [1200] LN2 Level Sensor and Control Faults ---
    E1200_SHA_LS_High_NotTriggered                : UDINT := 1200001; // SHA.LS high not reached
    E1201_SHB_LS_High_NotTriggered                : UDINT := 1200002; // SHB.LS high not reached
    E1202_SHC_LS_High_NotTriggered                : UDINT := 1200003; // SHC.LS high not reached
    E1203_SHA_LS_StuckLow                         : UDINT := 1200004; // SHA.LS low not clearing
    E1204_LevelSensor_HighDuringRefill            : UDINT := 1200005; // High level sensor triggered during fill
    E1205_LevelSensor_LowDuringIdle               : UDINT := 1200006; // Low level sensor triggered unexpectedly
	E1206_LN2_Level_ShutdownTimeout 			  : UDINT := 1200007; // Ln2 filling shutdown timeout: at least one LN2 filling ctrl still active.	
	E1207_LN2_ShutDown_V1_Failed				  : UDINT := 1200008; // LN2 Valve 1 failed to turn off
	E1208_LN2_ShutDown_V2_Failed				  : UDINT := 1200009; // LN2 Valve 2 failed to turn off
	E1209_LN2_ShutDown_V3_Failed  				  : UDINT := 1200010; // LN2 Valve 3 failed to turn off
    // --- [1300] Temperature Control Errors ---
    E1300_Temp_RadiationShieldNotReached          : UDINT := 1300001; // Shield temp > 120 K too long
    E1301_DetectorRampTooFast                     : UDINT := 1300002; // Detector cooled > 1 K/min
    E1302_T_CFO_Below85_NotControlled             : UDINT := 1300003; // T-CFO reached < 85K but control failed
    E1303_T_IMG_Below85_NotControlled             : UDINT := 1300004; // T-IMG reached < 85K but control failed
    E1304_CFO_ControlLoopInstability              : UDINT := 1300005; // CFO T-control oscillating
    E1305_IMG_ControlLoopInstability              : UDINT := 1300006; // IMG T-control oscillating
    E1306_ShieldTempRising                        : UDINT := 1300007; // Radiation shield temp rising after <100K
    E1307_EarFlange_TempFault                     : UDINT := 1300008; // Ear flange temp anomaly
	E1308_EarFlange_TempCtrlFault                 : UDINT := 1300009; // Ear flange heater or ctrl loop failure
    E1309_FieldRotator_TempFault                  : UDINT := 1300010; // Field rotator temp anomaly

    // --- [1400] Pressure Monitoring Errors ---
    E1400_VAG_PCB_TooHigh                         : UDINT := 1400001; // PCB pressure > 1 mbar
    E1401_VAG_PCA_TooHigh                         : UDINT := 1400002; // PCA pressure > 1 mbar
    E1402_VAG_PCB_PumpoutFailed                   : UDINT := 1400003; // PCB pressure > 0.1 mbar after pumpout
    E1403_VAG_PCA_PumpoutFailed                   : UDINT := 1400004; // PCA pressure > 0.1 mbar after pumpout
    E1404_VAG_A3_TooHigh                          : UDINT := 1400005; // A3 pressure > 0.1 mbar
    E1405_RepumpingRequired                       : UDINT := 1400006; // Re-pumping needed unexpectedly

    // --- [1500] Sequence Timing Errors ---
    E1500_CFO_ValveTimingError                    : UDINT := 1500001; // PCB.C1/2 sequence out of timing
    E1501_IMG_ValveTimingError                    : UDINT := 1500002; // PCA.C1/2 sequence out of timing
    E1502_PumpingOverlapDetected                  : UDINT := 1500003; // CFO + IMG connected to PVP A simultaneously
    E1503_EvaporationWaitTimeout                  : UDINT := 1500004; // 300s wait expired before safe pressure
    E1504_TempRampWaitTimeout                     : UDINT := 1500005; // Temp ramp timeout

    // --- [1600] Manual Intervention / Abort ---
    E1600_Operator_AbortedCooldown                : UDINT := 1600001; // Operator manually stopped cooldown
    E1601_Operator_AbortedFilling                 : UDINT := 1600002; // Operator stopped filling before LS high
    E1602_OperatorSwitchedPumpDuringFill          : UDINT := 1600003; // Pump config changed during fill

    // --- [1700] Pump Coordination Errors ---
    E1700_PVP_A_UsedInBothLoops                   : UDINT := 1700001; // Pump PVP A connected to both loops
    E1701_PVP_A_NotSwitchedBackToVacuum           : UDINT := 1700002; // PVP A not restored to vacuum system
    E1702_PVP_A_SwitchingTimeout                  : UDINT := 1700003; // Timeout during PVP A valve switch

    // --- [1800] Interlock Violations ---
    E1800_VentingValveOpenDuringCooldown          : UDINT := 1800001; // Venting valve is open during cooldown
    E1801_PCB_ValveOpen_Below80K                  : UDINT := 1800002; // PCB.C1/C2 open below 80 K
    E1802_PCA_ValveOpen_Below80K                  : UDINT := 1800003; // PCA.C1/C2 open below 80 K
    E1803_CooldownStartedBeforeShieldBelow120K    : UDINT := 1800004; // Started IMG/CFO cooldown too early

	// --- [1900] PTC Errors ---
	E1900_PTC1_NotInitialized					  : UDINT := 1900001; // PTC 1 not initialized
	E1901_PTC2_NotInitialized					  : UDINT := 1900002; // PTC 2 not initialized
	E1902_PTC3_NotInitialized					  : UDINT := 1900003; // PTC 3 not initialized
	E1903_PTC1_NotActive					  	  : UDINT := 1900004; // PTC 1 not Active
	E1904_PTC2_NotActive					  	  : UDINT := 1900005; // PTC 2 not Active
	E1905_PTC3_NotActive					  	  : UDINT := 1900006; // PTC 3 not Active
	
	E1906_PTC_Failure						  	  : UDINT := 1900007; // One or more PTCs failed
	E1907_PTC_ShutdownTimeout 					  : UDINT := 1900008; // PTC shutdown timeout: at least one PTC still active.

	// --- [2100] PTC Errors ---	
	E2101_StopCooldownPTCFailure 				  : UDINT := 2100001; // Max attempts to stop PTCs exceeded.
    E2102_StopCooldownLN2Failure 				  : UDINT := 2100002; // Max attempts to stop LN2 filling exceeded.
END_VAR


M_Configure();

M_ReadSensors();

M_ExecuteControllers();

// Early Refilling management
IF NOT bEarlyRefillDone THEN
	
    M_Manage_Early_Refilling();
	
END_IF

M_UpdateStatus(
				all_cryo_temps:= all_cryo_temps,
				all_heaters := all_heaters,
				all_t_ctrls := all_t_ctrls,
				all_t_votes := all_t_votes,
				interlocks := interlocks);

M_HandleEvents();

M_StateMachine(
				all_cryo_temps:= all_cryo_temps,
				all_heaters := all_heaters,
				all_t_ctrls := all_t_ctrls,
				all_t_votes := all_t_votes,
				interlocks := interlocks);


IF bReset_Valves THEN
	M_ResetValves();
	bReset_Valves := FALSE;
END_IF


IF in_Cryo_Stat.bWarmUpActive THEN
	M_Stop_PTCs_During_WarmUP();
END_IF


 
{IF defined (V2_SIM)}

M_Simulated_Sens_Acts();

{END_IF}

(* COOL_DOWN *)
METHOD M_Activity_Check_Preconditions
VAR_INPUT
END_VAR

// CHECK_COOL_DOWN_PRECONDITIONS

stat.bActive := TRUE;
stat.bDone := FALSE;



// --- Precondition Check: System in Vacuum ---
IF in_Cryo_Stat.bInGoodVacuum OR in_Cryo_Stat.bInVacuum THEN
		;
ELSE
	M_SetError(nCode := E1000_PressureTooHigh,
				sMessage := 'System pressure too high: p > 1e-4 mbar');
		
//    stat.nState := E_MET_CRYO_COOLDOWN_STATE.ERROR;
//    stat.sState := 'Error: Vacuum pressure is too high.';
    RETURN; 
END_IF

// --- Precondition Check: Warm UP Not Active ---
IF in_Cryo_Stat.bWarmUpActive THEN
	M_SetError(nCode:= E1001_WarmUpHeatersActive,
				sMessage := 'Warm-up heaters are active');

//    stat.nState := E_MET_CRYO_COOLDOWN_STATE.ERROR;
//    stat.sState := 'Error: Warm-Up is active.';
    RETURN; 
END_IF

// --- Precondition Check: Venting Valves Closed ---
IF NOT in_Cryo_Stat.bVentingValvesAreClosed THEN
		M_SetError(nCode:= E1003_VentingValveOpen,
				sMessage := 'Venting valves are open');
//    stat.nState := E_MET_CRYO_COOLDOWN_STATE.ERROR;
//    stat.sState := 'Error: Venting valves are not closed.';
    RETURN; 
END_IF

// --- Precondition Check: Regeneration Not Active ---
IF in_Cryo_Stat.bRegenerationActive THEN
		M_SetError(nCode:= E1002_SorptionHeaterActive,
				sMessage := 'Regeneration is active');
//    stat.nState := E_MET_CRYO_COOLDOWN_STATE.ERROR;
//    stat.sState := 'Error: Regeneration is active.';
    RETURN; 
END_IF

// --- Precondition Check: Pumps Running ---
IF NOT in_Cryo_Stat.bPumpsAreRunning THEN
		M_SetError(nCode:= E1004_PumpsNotRunning,
				sMessage := 'Pumps are Not running');
//    stat.nState := E_MET_CRYO_COOLDOWN_STATE.ERROR;
//    stat.sState := 'Error: Pumps are Not running.';
    RETURN; 
END_IF

// --- Precondition Check: Evacuation Stopped ---
IF NOT in_Cryo_Stat.bEvacuationActive THEN
		M_SetError(nCode:= E1006_EvacuationNotActive,
				sMessage := 'Evacuation Not Active');
//    stat.nState := E_MET_CRYO_COOLDOWN_STATE.ERROR;
//    stat.sState := 'Error: Evacuation Nor Active.';
    RETURN; 
END_IF

// --- Precondition Check: Cool Down Active ---
IF NOT bESO_LN2_Supply THEN
				M_SetError(nCode:= E1005_LN2SupplyNotReady,
				sMessage := 'LN2 supply not connected');
//    stat.nState := E_MET_CRYO_COOLDOWN_STATE.ERROR;
//    stat.sState := 'Error: LN2 supply not connected.';
    RETURN; 
END_IF


stat.nState := E_MET_CRYO_COOLDOWN_STATE.START_COOL_DOWN;
stat.sState := 'Preconditions met...';
END_METHOD

METHOD M_Activity_Cold_State : BOOL
VAR_INPUT
END_VAR
VAR_INST

	sFillTime:			STRING(16) := '11:00:00'; // UTC Time
	sCurrentTime:			STRING(16);
END_VAR
// 1. Check if filling is active

IF NOT lc_ln2_level_ctrl[1].bActive THEN
		ctrl.bEnable_LN2_Level_Control[1] := TRUE;
END_IF

IF NOT lc_ln2_level_ctrl[2].bActive THEN
		ctrl.bEnable_LN2_Level_Control[2] := TRUE;
END_IF

IF NOT lc_ln2_level_ctrl[3].bActive THEN
		ctrl.bEnable_LN2_Level_Control[3] := TRUE;
END_IF	



// Check if PTCs are active

IF NOT M_Check_PTCs_Status() THEN
	//RETURN;
	;
END_IF

// Start LN2 filling at specific time

sCurrentTime := F_TIME_HHMMSS();

IF sCurrentTime = sFillTime THEN
		
		lc_ln2_level_ctrl[1].M_Set_LN2FillingFlag();
		lc_ln2_level_ctrl[2].M_Set_LN2FillingFlag();
		lc_ln2_level_ctrl[3].M_Set_LN2FillingFlag();	
		logs.M_LogInfo(CONCAT('LN2 Filling started at:',F_TIME_HHMMSS()));	

END_IF
END_METHOD

METHOD M_Activity_Cool_Down_Finished : BOOL
VAR_INPUT
END_VAR
	

IF stat.bReadyForOperations THEN
	stat.bActive := FALSE;
	stat.bPermitEvacuationStop := TRUE;
	stat.sState := 'Cryostat Operational';
	logs.M_LogInfo('Cryostat ready for operations...');
	stat.bDone := TRUE;

ELSE
	logs.M_LogInfo('Cool_Down stopped: Not ready for operations');
	stat.bActive := FALSE;
	stat.bPermitEvacuationStop := FALSE;
	stat.bDone := FALSE;

END_IF

ctrl.bEnable := FALSE;

M_Activity_Cool_Down_Finished := TRUE;
stat.nState := E_MET_CRYO_COOLDOWN_STATE.NONE;
END_METHOD

METHOD M_Activity_Error_Handling
VAR_INPUT
END_VAR
stat.bError := TRUE;

IF ctrl.bReset THEN
    stat.nErrorCode := 0;
    stat.sErrorMessage := '';
    stat.sRecoverySuggestion := '';
    stat.nState := E_MET_CRYO_COOLDOWN_STATE.NONE;
    ctrl.bReset := FALSE;
	stat.bError := FALSE;
    RETURN;
END_IF

stat.nState := E_MET_CRYO_COOLDOWN_STATE.ERROR;

CASE stat.nErrorCode OF

//LN2 Shutdown Errors
E1206_LN2_Level_ShutdownTimeout:
    stat.sErrorMessage := 'LN2 shutdown timed out. One or more valves still active.';
    stat.sRecoverySuggestion := 'Check LN2 valve status and retry shutdown. Inspect hardware if needed.';
    
E1207_LN2_SHUTDOWN_V1_FAILED:
    stat.sErrorMessage := 'Valve 1 (Stiff Ring) failed to turn off.';
    stat.sRecoverySuggestion := 'Check valve actuator or control signal. Reset and retry.';

E1208_LN2_SHUTDOWN_V2_FAILED:
    stat.sErrorMessage := 'Valve 2 (Middle Segment) failed to turn off.';
    stat.sRecoverySuggestion := 'Inspect valve PCB.C2. Confirm it is not stuck or unresponsive.';

E1209_LN2_SHUTDOWN_V3_FAILED:
    stat.sErrorMessage := 'Valve 3 (Lower Segment) failed to turn off.';
    stat.sRecoverySuggestion := 'Inspect valve SHC.V and confirm signal reaches actuator.';

//PTC Errors 
E1903_PTC1_NotActive:
    stat.sErrorMessage := 'PTC 1 is not active during cooldown.';
    stat.sRecoverySuggestion := 'Try toggling PTC 1 via recovery. Check interlocks or initialization failure.';

E1904_PTC2_NotActive:
    stat.sErrorMessage := 'PTC 2 is not active.';
    stat.sRecoverySuggestion := 'Inspect PTC 2 enable logic. Confirm interlock and power status.';

E1905_PTC3_NotActive:
    stat.sErrorMessage := 'PTC 3 is not active.';
    stat.sRecoverySuggestion := 'Check if cooldown started too early or if PTC initialization failed.';

E1906_PTC_Failure:
    stat.sErrorMessage := 'PTC toggle recovery failed after timeout.';
    stat.sRecoverySuggestion := 'Verify power, control, and bActive flags of PTCs. Inspect fault registers.';

E2101_StopCooldownPTCFailure:
    stat.sErrorMessage := 'PTCs failed to stop after max attempts.';
    stat.sRecoverySuggestion := 'Manually inspect PTC status and confirm command interface is functional.';

//General Cooldown Control
E2102_StopCooldownLN2Failure:
    stat.sErrorMessage := 'LN2 filling control did not stop after max attempts.';
    stat.sRecoverySuggestion := 'Manually override LN2 level controller and check for persistent command signals.';

//future entries 
0:
    stat.sErrorMessage := '';
    stat.sRecoverySuggestion := '';

ELSE
	stat.sErrorMessage := 'Unknown error code';
    //stat.sErrorMessage := 'Unknown error code: ' + UDINT_TO_STRING(stat.nErrorCode);
    stat.sRecoverySuggestion := 'Refer to system logs and manual diagnostics.';
END_CASE
END_METHOD

METHOD M_Activity_Finished
VAR_INPUT
END_VAR
stat.nState := E_MET_CRYO_COOLDOWN_STATE.NONE;
stat.bActive := FALSE;
stat.bDone := TRUE;
END_METHOD

METHOD M_Activity_Keep_Cooling : BOOL
VAR_INPUT
END_VAR
VAR_IN_OUT
	{attribute 'OPC.UA.DA' := '0'}
	all_cryo_temps:					FB_METIS_TEMPERATURES;
	{attribute 'OPC.UA.DA' := '0'}
	all_heaters:					FB_METIS_HEATERS;
	{attribute 'OPC.UA.DA' := '0'}
	all_t_ctrls:      				FB_METIS_TCTRL;
	{attribute 'OPC.UA.DA' := '0'}
	all_t_votes: 					FB_METIS_VOTERS;
	{attribute 'OPC.UA.DA' := '0'}
	interlocks:						T_METIS_CRYO_INTERLOCKS;
END_VAR
//// IF Cool Down is not stopped manually 

IF NOT trigDisable.Q THEN
	
//		IF M_Activity_Start_LN2_Filling(
//						all_cryo_temps:= all_cryo_temps,
//						all_heaters := all_heaters,
//						all_t_ctrls := all_t_ctrls,
//						all_t_votes := all_t_votes,
//						interlocks := interlocks)
//		OR
//		 M_Standalone_LN2_Filling(
//									all_cryo_temps:= all_cryo_temps,
//									all_heaters := all_heaters,
//									all_t_ctrls := all_t_ctrls,
//									all_t_votes := all_t_votes,
//									interlocks := interlocks)
//		THEN
						
			// Check LN2 Filling Status
			IF NOT M_Check_LN2_Filling_Status() THEN
				//RETURN;
				; (*Once all valves are available, put return back*)
			END_IF			
						

//		ELSE
//					M_Standalone_LN2_Filling(
//									all_cryo_temps:= all_cryo_temps,
//									all_heaters := all_heaters,
//									all_t_ctrls := all_t_ctrls,
//									all_t_votes := all_t_votes,
//									interlocks := interlocks);
//		END_IF


	
	IF NOT M_Check_PTCs_Status() THEN
		//RETURN;
		;
	END_IF
	
	// TODO: Add other checks
	
	IF stat.bReadyForOperations THEN
		stat.nState := E_MET_CRYO_COOLDOWN_STATE.STOPPING_COOL_DOWN;
    	stat.sState := 'Cool down complete: Cryostat is operational';
    	logs.M_LogInfo('Cool down complete: Cryostat is operational');
	ELSE 
		stat.nState := E_MET_CRYO_COOLDOWN_STATE.KEEP_COOLING;
    	stat.sState := 'Cooling...';
		
	END_IF

ELSE
    stat.nState := E_MET_CRYO_COOLDOWN_STATE.STOPPING_COOL_DOWN;
    stat.sState := 'Cool down interrupted by operator';
    logs.M_LogInfo('Cool down interrupted by operator');
END_IF
END_METHOD

METHOD M_Activity_None
VAR_INPUT
END_VAR
VAR_IN_OUT
	{attribute 'OPC.UA.DA' := '0'}
	all_cryo_temps:					FB_METIS_TEMPERATURES;
	{attribute 'OPC.UA.DA' := '0'}
	all_heaters:					FB_METIS_HEATERS;
	{attribute 'OPC.UA.DA' := '0'}
	all_t_ctrls:      				FB_METIS_TCTRL;
	{attribute 'OPC.UA.DA' := '0'}
	all_t_votes: 					FB_METIS_VOTERS;
	{attribute 'OPC.UA.DA' := '0'}
	interlocks:						T_METIS_CRYO_INTERLOCKS;
END_VAR

stat.bActive := FALSE;
stat.bError  := FALSE;
stat.bPermitEvacuationStop := FALSE; // Evacuation is not allowed to stop

// Check enable and Interlocks
IF ctrl.bEnable AND NOT interlocks.bInterlock_CoolDown THEN
	stat.nState := E_MET_CRYO_COOLDOWN_STATE.CHECK_PRECONDITIONS;
ELSE
	stat.nState := E_MET_CRYO_COOLDOWN_STATE.NONE;
	stat.sState := 'Cool-Down OFF';
END_IF
END_METHOD

METHOD M_Activity_Start_Cool_Down : BOOL
VAR_INPUT
END_VAR
VAR_IN_OUT
	{attribute 'OPC.UA.DA' := '0'}
	all_cryo_temps:					FB_METIS_TEMPERATURES;
	{attribute 'OPC.UA.DA' := '0'}
	all_heaters:					FB_METIS_HEATERS;
	{attribute 'OPC.UA.DA' := '0'}
	all_t_ctrls:      				FB_METIS_TCTRL;
	{attribute 'OPC.UA.DA' := '0'}
	all_t_votes: 					FB_METIS_VOTERS;
	{attribute 'OPC.UA.DA' := '0'}
	interlocks:						T_METIS_CRYO_INTERLOCKS;
END_VAR
// TODO: Implement Handle interlocks
M_HandleInterlocks();

IF stat.bError THEN
    stat.sState := 'Interlocks not satisfied – aborting start';
    stat.nState := E_MET_CRYO_COOLDOWN_STATE.ERROR;
    RETURN;
END_IF

stat.bPermitEvacuationStop := FALSE; // Evacuation is not allowed to stop
stat.bActive := TRUE;
stat.bDone   := FALSE;

bEarlyRefillDone := FALSE;

//IF in_Cryo_Stat.lrRadiationShieldsTempK > in_lrRadShld_TempK_TO_Start_PTCs THEN
	
	stat.sState := 'Starting LN2 Filling...';
	stat.nState := E_MET_CRYO_COOLDOWN_STATE.START_FILLING_LN2;
	bStandaloneLN2Filling := FALSE;
//ELSE
//	bStandaloneLN2Filling := TRUE;	
//	stat.nState := E_MET_CRYO_COOLDOWN_STATE.START_PTCS;
//	stat.sState := 'Radiation shield temp achieved, preparing PTC start...';
//	logs.M_LogInfo('Radiation shield temp achieved, preparing PTC start...');
//END_IF
END_METHOD

METHOD M_Activity_Start_LN2_Filling : BOOL
VAR_INPUT
END_VAR
VAR_IN_OUT
	{attribute 'OPC.UA.DA' := '0'}
	all_cryo_temps:					FB_METIS_TEMPERATURES;
	{attribute 'OPC.UA.DA' := '0'}
	all_heaters:					FB_METIS_HEATERS;
	{attribute 'OPC.UA.DA' := '0'}
	all_t_ctrls:      				FB_METIS_TCTRL;
	{attribute 'OPC.UA.DA' := '0'}
	all_t_votes: 					FB_METIS_VOTERS;
	{attribute 'OPC.UA.DA' := '0'}
	interlocks:						T_METIS_CRYO_INTERLOCKS;
END_VAR
//VAR_INST
//	tDelaySHB:			TIME := T#900S;
//	tDelaySHC:			TIME := T#900S;
//	tDelaySHCold:		TIME := T#4H;
//END_VAR

// IF Cool Down is not stopped manually 

IF NOT trigDisable.Q THEN 
	
		CASE stat.nFillingState OF
	
		E_MET_CRYO_LN2_FILLING_STATE.NONE:

			stat.nFillingState := E_MET_CRYO_LN2_FILLING_STATE.CHECK_PRECONDITIONS; 
		
		(**** Preconditions check ****)
		
		E_MET_CRYO_LN2_FILLING_STATE.CHECK_PRECONDITIONS: 

			IF NOT in_Cryo_Stat.bEvacuationActive OR NOT in_Cryo_Stat.bPumpsAreRunning THEN
				M_SetError(E1004_PumpsNotRunning, 'Evacuation is not active');
				stat.nFillingState := E_MET_CRYO_LN2_FILLING_STATE.ERROR;
			ELSIF NOT bESO_LN2_Supply THEN
				M_SetError(E1005_LN2SupplyNotReady, 'LN2 Supply is not available');
				stat.nFillingState := E_MET_CRYO_LN2_FILLING_STATE.ERROR;
			ELSE
				stat.nFillingState := E_MET_CRYO_LN2_FILLING_STATE.START_LEVEL_CONTROL_SHA;
				ctrl.bEnable_LN2_Level_Control[1] := TRUE; // Enable SHA control
			END_IF
			
			// Reseting LN2 level control timeouts	
			tDelay_SHB(IN := FALSE);
			tDelay_SHC(IN := FALSE);
			tDelay_SHs_Cold(IN := FALSE);
			
			
			
		(**** Begin LN2 level control at SHA (Stiff Ring) ****)	
		
		E_MET_CRYO_LN2_FILLING_STATE.START_LEVEL_CONTROL_SHA:
		
			IF lc_ln2_level_ctrl[1].out_LN2_Level = E_METIS_CRYO_LN2_SENSOR_LEVELS.LOW OR 
				lc_ln2_level_ctrl[1].out_LN2_Level = E_METIS_CRYO_LN2_SENSOR_LEVELS.HIGH OR
				lc_ln2_level_ctrl[1].out_LN2_Level = E_METIS_CRYO_LN2_SENSOR_LEVELS.HIGH_ALARM THEN
				
				stat.nFillingState := E_MET_CRYO_LN2_FILLING_STATE.LEVEL_LOW_SHA;
				stat.sState := 'LN2 at or above low level at SHA';
			ELSE
				
				stat.sState := 'Filling Stiff Ring...';
							
			END_IF	
			IF ctrl.bReset THEN
				stat.nFillingState := E_MET_CRYO_LN2_FILLING_STATE.CHECK_PRECONDITIONS;
			END_IF	

		(**** LN2 reached low level at SHA ****)
		
		E_MET_CRYO_LN2_FILLING_STATE.LEVEL_LOW_SHA:
			
			tDelay_SHC(IN := TRUE, PT := tDelaySHC);
			IF tDelay_SHC.Q THEN
				// Start Bottom Segment Fill (SHC)
				ctrl.bEnable_LN2_Level_Control[3] := TRUE;
				stat.sState := 'Filling Bottom Segment...';
				stat.nFillingState := E_MET_CRYO_LN2_FILLING_STATE.START_LEVEL_CONTROL_SHC;
				tDelay_SHC(IN := FALSE);
			ELSE
				stat.sState := CONCAT('LN2 low level at SHA. SHC start timeout: ',
							 F_TON_TO_TIME_STRING(Timer := tDelay_SHC));
			END_IF
			IF ctrl.bReset THEN
				stat.nFillingState := E_MET_CRYO_LN2_FILLING_STATE.CHECK_PRECONDITIONS;
			END_IF
			
		(**** Begin LN2 control at SHC (Bottom Segment) ****)			
			
		E_MET_CRYO_LN2_FILLING_STATE.START_LEVEL_CONTROL_SHC:

			IF lc_ln2_level_ctrl[3].out_LN2_Level = E_METIS_CRYO_LN2_SENSOR_LEVELS.LOW OR 
				lc_ln2_level_ctrl[3].out_LN2_Level = E_METIS_CRYO_LN2_SENSOR_LEVELS.HIGH OR
				lc_ln2_level_ctrl[3].out_LN2_Level = E_METIS_CRYO_LN2_SENSOR_LEVELS.HIGH_ALARM THEN
				
				stat.nFillingState := E_MET_CRYO_LN2_FILLING_STATE.LEVEL_LOW_SHC;
				stat.sState := 'LN2 at or above low level at SHC';
			ELSE
				
				stat.sState := 'Filling Stiff Ring + Bottom segment...';
							
			END_IF
			IF ctrl.bReset THEN
				stat.nFillingState := E_MET_CRYO_LN2_FILLING_STATE.CHECK_PRECONDITIONS;
			END_IF
			
		(**** LN2 reached low level at SHC ****)

		E_MET_CRYO_LN2_FILLING_STATE.LEVEL_LOW_SHC:

			tDelay_SHB(IN := TRUE, PT := tDelaySHB);
			IF tDelay_SHB.Q THEN

				stat.nFillingState := E_MET_CRYO_LN2_FILLING_STATE.START_LEVEL_CONTROL_SHB;
				tDelay_SHB(IN := FALSE);
			ELSE
				stat.sState := CONCAT('LN2 low level at SHC. SHB start timeout: ',
							 F_TON_TO_TIME_STRING(Timer := tDelay_SHB));
			END_IF
			IF ctrl.bReset THEN
				stat.nFillingState := E_MET_CRYO_LN2_FILLING_STATE.CHECK_PRECONDITIONS;
			END_IF

		(**** Begin LN2 control at SHB (Middle Segment) ****)	
			
		E_MET_CRYO_LN2_FILLING_STATE.START_LEVEL_CONTROL_SHB:
		
			// Start Middle Segment Fill (SHB)
			ctrl.bEnable_LN2_Level_Control[2] := TRUE;
			stat.sState := 'Filling Middle Segment...';
			stat.nFillingState := E_MET_CRYO_LN2_FILLING_STATE.FILLING;
			
			IF ctrl.bReset THEN
				stat.nFillingState := E_MET_CRYO_LN2_FILLING_STATE.CHECK_PRECONDITIONS;
			END_IF

		(**** Actively filling LN2 (steady operation) ****)
		
		E_MET_CRYO_LN2_FILLING_STATE.FILLING:
		
			IF NOT in_Cryo_Stat.bEvacuationActive THEN
				M_SetError(E1004_PumpsNotRunning, 'Evacuation is not active');
				stat.nFillingState := E_MET_CRYO_LN2_FILLING_STATE.ERROR;
			ELSIF NOT bESO_LN2_Supply THEN
				M_SetError(E1005_LN2SupplyNotReady, 'LN2 Supply is not available');
				stat.nFillingState := E_MET_CRYO_LN2_FILLING_STATE.ERROR;
			ELSE
				
				IF in_Cryo_Stat.lrRadiationShieldsTempK > in_lrRadShld_TempK_TO_Start_PTCs THEN
					stat.sState := CONCAT('Filling All Vessels – Waiting Shields Temp <', LREAL_TO_STRING(in_lrRadShld_TempK_TO_Start_PTCs));
//					IF NOT M_Check_LN2_Filling_Status() THEN
//						RETURN; // Error detected or recovery in progress
//					END_IF

				ELSE
						stat.nFillingState := E_MET_CRYO_LN2_FILLING_STATE.RADIATION_SHIELDS_COLD;
				END_IF

				IF ctrl.bReset THEN
					stat.nFillingState := E_MET_CRYO_LN2_FILLING_STATE.CHECK_PRECONDITIONS;
				END_IF					
			
			END_IF

		(**** Shield are COLD enough, Wait 4 hours****)			
			
		E_MET_CRYO_LN2_FILLING_STATE.RADIATION_SHIELDS_COLD:
				
				tDelay_SHs_Cold(IN := TRUE, PT := tDelaySHCold);
				
				IF tDelay_SHs_Cold.Q THEN
					stat.nFillingState := E_MET_CRYO_LN2_FILLING_STATE.START_PTCS;
					tDelay_SHs_Cold(IN := FALSE, PT := tDelaySHCold); // RESET timer
				ELSE
					stat.sState := CONCAT('Shield segments are COLD. PTCs start timeout: ',
							 F_TON_TO_TIME_STRING(Timer := tDelay_SHs_Cold));
					IF ctrl.bReset THEN
						stat.nFillingState := E_MET_CRYO_LN2_FILLING_STATE.CHECK_PRECONDITIONS;
					END_IF
//					IF NOT M_Check_LN2_Filling_Status() THEN
//						RETURN; // Error detected or recovery in progress
//					END_IF

					
				END_IF				

				
		(**** Transition to PTC start ****)	
		
		E_MET_CRYO_LN2_FILLING_STATE.START_PTCS:
		
				stat.nState := E_MET_CRYO_COOLDOWN_STATE.START_PTCS;
				stat.sState := 'Radiation shield temp achieved, preparing PTC start...';
				logs.M_LogInfo('Radiation shield temp achieved, preparing PTC start...');
				M_Activity_Start_LN2_Filling := TRUE; // Allow sequence to continue
				
				IF ctrl.bReset THEN
					stat.nFillingState := E_MET_CRYO_LN2_FILLING_STATE.CHECK_PRECONDITIONS;
				END_IF
		
	
		E_MET_CRYO_LN2_FILLING_STATE.ERROR: // Error Handling / Safe Shutdown
			IF ctrl.bReset THEN
				stat.nFillingState := E_MET_CRYO_LN2_FILLING_STATE.CHECK_PRECONDITIONS;
			END_IF
			IF NOT M_Check_LN2_Filling_Status() THEN
				RETURN; // Error detected or recovery in progress
			END_IF
			// Optional: auto-reset if conditions restored
			IF in_Cryo_Stat.bEvacuationActive AND bESO_LN2_Supply THEN
				stat.nFillingState := E_MET_CRYO_LN2_FILLING_STATE.CHECK_PRECONDITIONS;
			END_IF
	
		END_CASE

ELSE
	stat.nFillingState := E_MET_CRYO_LN2_FILLING_STATE.CHECK_PRECONDITIONS;
	ctrl.bEnable_LN2_Level_Control[1] := FALSE;
	ctrl.bEnable_LN2_Level_Control[2] := FALSE;
	ctrl.bEnable_LN2_Level_Control[3] := FALSE;
	
	tDelay_SHB(IN := FALSE);
	tDelay_SHC(IN := FALSE);
	tDelay_SHs_Cold(IN := FALSE);
	
	M_Activity_Stop_LN2_Filling();

	stat.nState := E_MET_CRYO_COOLDOWN_STATE.STOPPING_COOL_DOWN;
	stat.sState := 'COOL_DOWN interrupted by operator...';
	logs.M_LogInfo('COOL_DOWN interrupted by operator...');
END_IF
END_METHOD

METHOD M_Activity_Start_PTCs : BOOL
VAR_INPUT
END_VAR
VAR_IN_OUT
	{attribute 'OPC.UA.DA' := '0'}
	all_cryo_temps:					FB_METIS_TEMPERATURES;
	{attribute 'OPC.UA.DA' := '0'}
	all_heaters:					FB_METIS_HEATERS;
	{attribute 'OPC.UA.DA' := '0'}
	all_t_ctrls:      				FB_METIS_TCTRL;
	{attribute 'OPC.UA.DA' := '0'}
	all_t_votes: 					FB_METIS_VOTERS;
	{attribute 'OPC.UA.DA' := '0'}
	interlocks:						T_METIS_CRYO_INTERLOCKS;
END_VAR

IF NOT trigDisable.Q THEN
	
//	IF M_Activity_Start_LN2_Filling(
//						all_cryo_temps:= all_cryo_temps,
//						all_heaters := all_heaters,
//						all_t_ctrls := all_t_ctrls,
//						all_t_votes := all_t_votes,
//						interlocks := interlocks)
//		OR
//		 M_Standalone_LN2_Filling(
//									all_cryo_temps:= all_cryo_temps,
//									all_heaters := all_heaters,
//									all_t_ctrls := all_t_ctrls,
//									all_t_votes := all_t_votes,
//									interlocks := interlocks)
//		THEN
						
		// Check LN2 Filling Status
			IF NOT M_Check_LN2_Filling_Status() THEN
				//RETURN;
				; (*Once all valves are available, put return back*)
			END_IF			
						

//		ELSE
//					M_Standalone_LN2_Filling(
//									all_cryo_temps:= all_cryo_temps,
//									all_heaters := all_heaters,
//									all_t_ctrls := all_t_ctrls,
//									all_t_votes := all_t_votes,
//									interlocks := interlocks);
//		END_IF
	
	IF bAllowPTCsStart THEN
		
	
		CASE stat.nPTCStartingState OF
	
		0: // Start delay for PTC 1
			IF ptc[1].stat.bInitialised THEN
				tDelayPTC_1(IN := TRUE, PT := T#10S);
				stat.sState := 'Waiting before enabling PTC 1...';
				stat.nPTCStartingState := 1;
			ELSE
				M_SetError(E1900_PTC1_NotInitialized, 'PTC 1 not initialized');
				logs.M_LogInfo('PTC 1 not initialized');
				stat.sState := 'PTC 1 not initialized';
				stat.nPTCStartingState := 1;
			END_IF
	
		1: // Enable PTC 1
			tDelayPTC_1(IN := TRUE, PT := T#10S);
			IF tDelayPTC_1.Q AND ptc[1].stat.bInitialised THEN
				//ptc[1].in_bEnable := TRUE;
				ctrl.bPTC_1_Enable := TRUE;
				tDelayPTC_2(IN := TRUE, PT := tDelayPTCStart);
				stat.sState := 'PTC 1 enabled, delaying for PTC 2...';
				stat.nPTCStartingState := 2;
			ELSE
				M_SetError(E1900_PTC1_NotInitialized, 'PTC 1 not initialized');
				logs.M_LogInfo('PTC 1 not initialized');
				stat.sState := 'PTC 1 not initialized';
				stat.nPTCStartingState := 2;
			END_IF
	
		2: // Enable PTC 2
			tDelayPTC_2(IN := TRUE, PT := tDelayPTCStart);
			IF ptc[2].stat.bInitialised THEN
				IF tDelayPTC_2.Q THEN
					ctrl.bPTC_2_Enable := TRUE;
					tDelayPTC_3(IN := TRUE, PT := tDelayPTCStart);
					stat.sState := 'PTC 2 enabled, delaying for PTC 3...';
					stat.nPTCStartingState := 3;
				END_IF
			ELSE
				M_SetError(E1901_PTC2_NotInitialized, 'PTC 2 not initialized');
				logs.M_LogInfo('PTC 2 not initialized');
				stat.sState := 'PTC 2 not initialized';
				stat.nPTCStartingState := 3;
			END_IF
	
		3: // Enable PTC 3
			tDelayPTC_3(IN := TRUE, PT := tDelayPTCStart);
			IF ptc[3].stat.bInitialised THEN
				IF tDelayPTC_3.Q THEN
					ctrl.bPTC_3_Enable := TRUE;
					stat.sState := 'PTCs enabled. Proceeding to temperature control.';
					stat.nPTCStartingState := 0;
					stat.nState := E_MET_CRYO_COOLDOWN_STATE.START_TEMP_CTRL_PTC;
					M_Activity_Start_PTCs := TRUE;
					RETURN;
				END_IF
			ELSE
				M_SetError(E1902_PTC3_NotInitialized, 'PTC 3 not initialized');
				logs.M_LogInfo('PTC 3 not initialized');
				stat.sState := 'PTC 3 not initialized';
				stat.nPTCStartingState := 4; 
			END_IF
		4:
			IF ptc[1].stat.bSystemOn OR ptc[2].stat.bSystemOn OR ptc[2].stat.bSystemOn THEN
					stat.nPTCStartingState := 0;
					stat.nState := E_MET_CRYO_COOLDOWN_STATE.START_TEMP_CTRL_PTC;
					logs.M_LogInfo('One or more PTCs enabled. Proceeding to temperature control.');
					M_Activity_Start_PTCs := TRUE;
			END_IF
	
		99: // Error fallback
	
			tDelayPTC_1(IN := FALSE);
			tDelayPTC_2(IN := FALSE);
			tDelayPTC_3(IN := FALSE);
			stat.sState := 'Error starting PTCs';
			bAllowPTCsStart := FALSE;
			stat.nPTCStartingState := 0; 
			stat.nState := E_MET_CRYO_COOLDOWN_STATE.START_PTCS;
			
		END_CASE
	
	ELSE
		stat.sState := 'Allow to start PTCs';
	END_IF
		
		
ELSE
	bAllowPTCsStart := FALSE;
	stat.nPTCStartingState := 0;
	tDelayPTC_1(IN := FALSE);
	tDelayPTC_2(IN := FALSE);
	tDelayPTC_3(IN := FALSE);
    stat.nState := E_MET_CRYO_COOLDOWN_STATE.STOPPING_COOL_DOWN;
    stat.sState := 'Cool down interrupted by operator';
    logs.M_LogInfo('Cool down interrupted by operator');
END_IF
END_METHOD

METHOD M_Activity_Start_Temp_Ctrl_PTC : BOOL
VAR_INPUT
END_VAR
VAR_IN_OUT
	{attribute 'OPC.UA.DA' := '0'}
	all_cryo_temps:					FB_METIS_TEMPERATURES;
	{attribute 'OPC.UA.DA' := '0'}
	all_heaters:					FB_METIS_HEATERS;
	{attribute 'OPC.UA.DA' := '0'}
	all_t_ctrls:      				FB_METIS_TCTRL;
	{attribute 'OPC.UA.DA' := '0'}
	all_t_votes: 					FB_METIS_VOTERS;
	{attribute 'OPC.UA.DA' := '0'}
	interlocks:						T_METIS_CRYO_INTERLOCKS;
END_VAR
//// IF Cool Down is not stopped manually 

IF NOT trigDisable.Q THEN
	
//		IF M_Activity_Start_LN2_Filling(
//						all_cryo_temps:= all_cryo_temps,
//						all_heaters := all_heaters,
//						all_t_ctrls := all_t_ctrls,
//						all_t_votes := all_t_votes,
//						interlocks := interlocks)
//		OR
//		 M_Standalone_LN2_Filling(
//									all_cryo_temps:= all_cryo_temps,
//									all_heaters := all_heaters,
//									all_t_ctrls := all_t_ctrls,
//									all_t_votes := all_t_votes,
//									interlocks := interlocks)
//		THEN
						
			// Check LN2 Filling Status
			IF NOT M_Check_LN2_Filling_Status() THEN
				//RETURN;
				; (*Once all valves are available, put return back*)
			END_IF			
						

//		ELSE
//					M_Standalone_LN2_Filling(
//									all_cryo_temps:= all_cryo_temps,
//									all_heaters := all_heaters,
//									all_t_ctrls := all_t_ctrls,
//									all_t_votes := all_t_votes,
//									interlocks := interlocks);
//		END_IF

	// Enable 3 heaters on three PTCs and one temp control loop to control them
	
	all_heaters.h_cry_pta.M_SetEnable();
	all_heaters.h_cry_ptb.M_SetEnable();
	all_heaters.h_cry_ptc.M_SetEnable();

	
	all_t_ctrls.tc_cry_pt.M_SetEnable();

	all_t_ctrls.tc_cry_pt.M_Set_SetPoint(
		m_eSetpointType := E_METIS_CTRL_SETPOINT_SWITCH.FIXED,
		m_lrFixedSetpoint := 40,
		m_lrSetpointOffset := 0.0, 
		m_pSetpointTemp := all_cryo_temps.M_SetTemperatureSensor(0));
		
	stat.nState := E_MET_CRYO_COOLDOWN_STATE.KEEP_COOLING;	

ELSE
    stat.nState := E_MET_CRYO_COOLDOWN_STATE.STOPPING_COOL_DOWN;
    stat.sState := 'Cool down interrupted by operator';
    logs.M_LogInfo('Cool down interrupted by operator');
END_IF
END_METHOD

METHOD M_Activity_Stop_LN2_Filling : BOOL
VAR_INPUT
END_VAR
VAR_INST
    bErrorCond            : BOOL := FALSE;
    bAttemptingTurnOFF    : BOOL := FALSE;

    TurningOFFTimeout     : TON;
    tTurningOFFTime       : TIME := T#2M;
END_VAR
// --- Step 1: Initiate shutdown only once
IF NOT bAttemptingTurnOFF THEN
    bAttemptingTurnOFF := TRUE;
    logs.M_LogInfo('Initiating LN2 filling shutdown...');
    
    TurningOFFTimeout(IN := TRUE, PT := tTurningOFFTime);

    ctrl.bEnable_LN2_Level_Control[1] := FALSE;
    ctrl.bEnable_LN2_Level_Control[2] := FALSE;
    ctrl.bEnable_LN2_Level_Control[3] := FALSE;
END_IF

// --- Step 2: Monitor shutdown progress
IF NOT TurningOFFTimeout.Q THEN
    IF lc_ln2_level_ctrl[1].LN2_Valve.stat.bActive
    OR lc_ln2_level_ctrl[2].LN2_Valve.stat.bActive
    OR lc_ln2_level_ctrl[3].LN2_Valve.stat.bActive THEN
        M_Activity_Stop_LN2_Filling := FALSE;
        RETURN;
    END_IF

